// TwinCAT 3 PLC project Plc_CHALET_Xts
// Title: CHALET_Xts
// Company: Beckhoff CH
// ProjectVersion: 4.2.1
// ProgramVersion: 3.1.4023.0
// libraries:
//   CHALET_BaseComponents, * (Beckhoff CH)
//   CHALET_Nc, * (Beckhoff CH)
//   Tc2_EtherCAT, * (Beckhoff Automation GmbH)
//   Tc2_Math, * (Beckhoff Automation GmbH)
//   Tc2_MC2, * (Beckhoff Automation GmbH)
//   Tc2_Standard, * (Beckhoff Automation GmbH)
//   Tc2_System, * (Beckhoff Automation GmbH)
//   Tc3_EventLogger, * (Beckhoff Automation GmbH)
//   Tc3_Mc3Definitions, * (Beckhoff Automation GmbH)
//   Tc3_McCollisionAvoidance, * (Beckhoff Automation GmbH)
//   Tc3_McCoordinatedMotion, * (Beckhoff Automation GmbH)
//   Tc3_Module, * (Beckhoff Automation GmbH)
//   Tc3_XTS_Utility, * (Beckhoff Automation GmbH)
// project tree:
//   COMPENENTs/Casting/ ToMover.TcPOU, ToGroup.TcPOU, ToMover_PLC.TcPOU, ToStation_PLC.TcPOU, ToTrigger.TcPOU, ToEnvironment.TcPOU, ToStation.TcPOU
//   COMPENENTs/ Class Diagram.TcCD (not stored)
//   COMPENENTs/Environment/ FB_XTS_Environment.TcPOU, I_XTS_Environment.TcIO
//   COMPENENTs/Group/ E_NcGroupCommands.TcDUT, FB_XTS_Group.TcPOU, I_XTS_Group.TcIO
//   COMPENENTs/Lubrication/ E_LubricationMode.TcDUT, E_SystemType.TcTLEO, FB_LubricationXTS.TcPOU
//   COMPENENTs/Mover/ FB_XTS_Axis.TcPOU, FB_XTS_Mover.TcPOU, I_XTS_Axis.TcIO, I_XTS_Mover.TcIO, I_XTS_Mover_PLC.TcIO
//   COMPENENTs/Mover/ProductData/ FB_XTS_ProductData.TcPOU, I_XTS_ProductData.TcIO
//   COMPENENTs/Station/ FB_XTS_Station.TcPOU, I_XTS_Station.TcIO, I_XTS_Station_PLC.TcIO
//   COMPENENTs/System/ FB_XTS_System.TcPOU, I_XTS_System_PLC.TcIO, I_XTS_System_Registration.TcIO
//   COMPENENTs/Trigger/ FB_XTS_Trigger.TcPOU, I_XTS_Trigger.TcIO
//   COMPENENTs/Zone/ FB_XTS_Zone.TcPOU, I_XTS_Zone.TcIO
//   Diag/ FB_XtsEtherCatDiag.TcPOU, ST_XtsMotorEtherCatDiag.TcDUT
//   FUNCTIONs/ F_BuildLogString.TcPOU, F_GetDistToPosModulo.TcPOU, F_InLimitTest.TcPOU
//   / XtsParameterlist.TcGVL

// ---- COMPENENTs/Group/E_NcGroupCommands.TcDUT
{attribute 'qualified_only'}
{attribute 'strict'}
{attribute 'to_string'}
TYPE E_NcGroupCommands :
(
	None:=0,
	GroupDisable:=150,
	GroupEnable,
	GroupReset,
	AddAxisListToGroup,
	RemoveAxisFromGroup,
	UngroupAllAxes
);
END_TYPE

// ---- COMPENENTs/Lubrication/E_LubricationMode.TcDUT
{attribute 'qualified_only'}
TYPE E_LubricationMode :
(
	TimeBased,
	DistanceBased,
	Continous
);
END_TYPE

// ---- COMPENENTs/Lubrication/E_SystemType.TcTLEO
{attribute 'qualified_only'}
TYPE E_SystemType :
(
 	BekaPico,
	SkfETP2WZ
);
END_TYPE

// ---- Diag/ST_XtsMotorEtherCatDiag.TcDUT
TYPE ST_XtsMotorEtherCatDiag :
STRUCT
	fbSource : FB_TcSourceInfo;
	fbAlarmNotInOpMode : FB_TcAlarm;
	fbAlarmNoCommunication : FB_TcAlarm;
	
	fbGetSlaveState : FB_EcGetSlaveState;
	nLastState : BYTE;
END_STRUCT
END_TYPE

// ---- XtsParameterlist.TcGVL
{attribute 'qualified_only'}
VAR_GLOBAL CONSTANT
	
	(*Checks whether the TC3 event logger is set as standard in the XTS prosessing unit.*)
	B_MSG_IF_TC3EVENTLOGGER_IS_NOT_DEFAULT: BOOL := TRUE;	

	MAX_MOVER_PER_SYSTEM : UINT := 50;
	MAX_MOTORS_PER_SYSTEM : UINT := 100;
	STATISTIC_AVG_PERIOD : TIME := T#10S;
END_VAR

// ---- COMPENENTs/Environment/I_XTS_Environment.TcIO
INTERFACE I_XTS_Environment  EXTENDS I_CH_Object

{attribute 'monitoring':='call'}
PROPERTY HR : HRESULT
GET
END_GET
END_PROPERTY

METHOD Initialize : HRESULT
END_METHOD

{attribute 'monitoring':='call'}
PROPERTY TrackIsRing : BOOL
GET
END_GET
END_PROPERTY

{attribute 'monitoring':='call'}
PROPERTY TrackLength : LREAL
GET
END_GET
END_PROPERTY

METHOD Update : HRESULT
VAR_INPUT
END_VAR
END_METHOD

PROPERTY UtilityEnvirement : Tc3_XTS_Utility.i_TcIoXtsEnvironment
GET
END_GET
END_PROPERTY

END_INTERFACE

// ---- COMPENENTs/Group/I_XTS_Group.TcIO
INTERFACE I_XTS_Group  EXTENDS I_CH_Object

METHOD AddAxisListToGroup : HRESULT
VAR_INPUT
	ipMovers : I_CH_List;
END_VAR
END_METHOD

METHOD AddingAxisToGroup : HRESULT
END_METHOD

PROPERTY AllAxesStanding : Bool
GET
END_GET
END_PROPERTY

METHOD ChangeGapMode : HRESULT
VAR_INPUT
	bFast : BOOL;
END_VAR
END_METHOD

METHOD Disable : HRESULT
VAR_INPUT
END_VAR
END_METHOD

METHOD Enable : HRESULT
VAR_INPUT
END_VAR
END_METHOD

{attribute 'monitoring':='call'}
PROPERTY GroupEnabled : BOOL
GET
END_GET
END_PROPERTY

{attribute 'monitoring':='call'}
PROPERTY HR : HRESULT
GET
END_GET
END_PROPERTY

METHOD Initialize : HRESULT
VAR_INPUT
END_VAR
END_METHOD

METHOD RemoveAxisFromGroup : HRESULT
VAR_INPUT
	ipMover : I_XTS_Mover;
END_VAR
END_METHOD

METHOD Reset : HRESULT
VAR_INPUT
END_VAR
END_METHOD

METHOD UngroupAllAxes : HRESULT
VAR_INPUT
END_VAR
END_METHOD

METHOD Update : HRESULT
VAR_INPUT
END_VAR
END_METHOD

{attribute 'monitoring':='call'}
PROPERTY UtilityCAGroup : I_Mc2CaGroup
GET
END_GET
END_PROPERTY

END_INTERFACE

// ---- COMPENENTs/Mover/I_XTS_Axis.TcIO
INTERFACE I_XTS_Axis EXTENDS CHALET_Nc.I_NcAxis_PLC

METHOD HaltCA : I_CH_Feedback
VAR_INPUT
	fDeceleration          : LREAL;
    fJerk                  : LREAL;
    fGap                   : LREAL;
END_VAR
END_METHOD

{attribute 'TcRpcEnable':='1'} //call methode via OPC-UA conection
METHOD MoveAbsoluteCA  : I_CH_Feedback
VAR_INPUT
	fPosition		: LREAL;
	
	(* This value determines the minimum gap to the predecessor for Collision Avoidance. *)
	fGap			: LREAL;
	
	(* Use the default dynamics if input=0. 
	The default dynamics can be read and written via property and is initialized with the default values in the NC parameter list. *)
	fVelocity		: LREAL;
	
	(* Use the default dynamics if input=0. 
	The default dynamics can be read and written via property and is initialized with the default values in the NC parameter list. *)
	fAcceleration	: LREAL;
	
	(* Use the default dynamics if input=0. 
	The default dynamics can be read and written via property and is initialized with the default values in the NC parameter list. *)
	fDeceleration	: LREAL;
	
	(* Use the default dynamics if input=0. 
	The default dynamics can be read and written via property and is initialized with the default values in the NC parameter list. *)
	fJerk			: LREAL;
	
	(* Defines the direction of the movement (e.g. for a modulo axis). 
		input=0 = mcDirectionNonModulo*)
	eDirection	: Tc3_Mc3Definitions.MC_DIRECTION;
	
	(* Use the Aborting mode without buffering if input=0. 
	BufferModes:
		-MC_Aborting: Default mode without buffering. The command is executed immediately and interrupts any other command that may be running.
		-MC_Buffered: The command is executed once no other command is running on the axis. The previous movement continues until it has stopped. The following command is started from standstill. *)
	eBufferMode   : Tc3_Mc3Definitions.MC_BUFFER_MODE;
END_VAR
END_METHOD

END_INTERFACE

// ---- COMPENENTs/Mover/I_XTS_Mover.TcIO
INTERFACE I_XTS_Mover EXTENDS I_CH_Object

{attribute 'OPC.UA.DA.Property' := '1'}
{attribute 'monitoring':='call'}
PROPERTY Coupled : BOOL
GET
END_GET
END_PROPERTY

METHOD Disable : HRESULT
VAR_INPUT
END_VAR
END_METHOD

{attribute 'monitoring':='call'}
PROPERTY DrivenDistance : LREAL
GET
END_GET
END_PROPERTY

METHOD Enable : HRESULT
VAR_INPUT
END_VAR
END_METHOD

{attribute 'OPC.UA.DA.Property' := '1'}
{attribute 'monitoring':='call'}
PROPERTY Feedback : I_CH_Feedback
GET
END_GET
END_PROPERTY

PROPERTY getAxisRef : REFERENCE TO Tc2_MC2.AXIS_REF
GET
END_GET
END_PROPERTY

METHOD HaltCA : HRESULT
VAR_INPUT
END_VAR
END_METHOD

{attribute 'monitoring':='call'}
PROPERTY IdentInGroup : IDENT_IN_GROUP_REF
GET
END_GET
END_PROPERTY

{attribute 'monitoring':='call'}
PROPERTY LagDistance : LREAL
GET
END_GET
END_PROPERTY

{attribute 'monitoring':='call'}
PROPERTY LastCmdTargedGap : LREAL
GET
END_GET
END_PROPERTY

{attribute 'monitoring':='call'}
PROPERTY LastCmdTargedPosition : LREAL
GET
END_GET
END_PROPERTY

{attribute 'monitoring':='call'}
PROPERTY LastCmdTargedVelocity : LREAL
GET
END_GET
END_PROPERTY

METHOD MoveAbsCA : HRESULT
VAR_INPUT
    fPosition              : LREAL;
    fVelocity              : LREAL;
    fGap                   : LREAL;
    eDirection             : Tc3_Mc3Definitions.MC_DIRECTION;
END_VAR
END_METHOD

{attribute 'monitoring':='call'}
PROPERTY MoverInGroup : BOOL
GET
END_GET
SET
END_SET
END_PROPERTY

{attribute 'OPC.UA.DA.Property' := '1'}
{attribute 'monitoring':='call'}
PROPERTY Moving : BOOL
GET
END_GET
END_PROPERTY

{attribute 'monitoring':='call'}
PROPERTY NextMover : I_XTS_Mover
GET
END_GET
END_PROPERTY

{attribute 'monitoring':='call'}
PROPERTY OID : OTCID
GET
END_GET
END_PROPERTY

{attribute 'monitoring':='call'}
PROPERTY ParentStation : I_XTS_Station
GET
END_GET
SET
END_SET
END_PROPERTY

{attribute 'monitoring':='call'}
PROPERTY PositionOnTrack : LREAL
GET
END_GET
END_PROPERTY

METHOD Reset : HRESULT
VAR_INPUT
END_VAR
END_METHOD

{attribute 'monitoring':='call'}
PROPERTY SetAcceleration : LREAL
GET
END_GET
END_PROPERTY

{attribute 'monitoring':='call'}
PROPERTY SetVelocity : LREAL
GET
END_GET
END_PROPERTY

{attribute 'monitoring':='call'}
PROPERTY TargedStation : STRING
GET
END_GET
SET
END_SET
END_PROPERTY

{attribute 'monitoring':='call'}
PROPERTY UtilityMover : I_TcIoXtsXpuMover
GET
END_GET
END_PROPERTY

END_INTERFACE

// ---- COMPENENTs/Mover/I_XTS_Mover_PLC.TcIO
INTERFACE I_XTS_Mover_PLC EXTENDS I_CH_Object

{attribute 'OPC.UA.DA.Property' := '1'}
{attribute 'monitoring':='call'}
PROPERTY DefaultAcceleration : LREAL
GET
END_GET
SET
END_SET
END_PROPERTY

{attribute 'OPC.UA.DA.Property' := '1'}
{attribute 'monitoring':='call'}
PROPERTY DefaultDeceleration : LREAL
GET
END_GET
SET
END_SET
END_PROPERTY

{attribute 'OPC.UA.DA.Property' := '1'}
{attribute 'monitoring':='call'}
PROPERTY DefaultJerk : LREAL
GET
END_GET
SET
END_SET
END_PROPERTY

{attribute 'monitoring':='call'}
PROPERTY DrivenDistance : LREAL
GET
END_GET
END_PROPERTY

(*The _ PLC interface provides the user with a simplified interface for commanding between the stations. Sometimes, however, this is not enough. 
Either you get the corresponding interface with the __Queryinterface or you can get full access with this property.*)
PROPERTY FullAccess : I_XTS_Mover
GET
END_GET
END_PROPERTY

{attribute 'monitoring':='call'}
PROPERTY LagDistance : LREAL
GET
END_GET
END_PROPERTY

{attribute 'monitoring':='call'}
PROPERTY LastCmdTargedGap : LREAL
GET
END_GET
END_PROPERTY

{attribute 'monitoring':='call'}
PROPERTY LUID : STRING
GET
END_GET
END_PROPERTY

//Returns the ID of the mover.
{attribute 'monitoring':='call'}
PROPERTY MoverID : STRING(3)
GET
END_GET
END_PROPERTY

{attribute 'monitoring':='call'}
PROPERTY NameXtsMover : STRING
GET
END_GET
END_PROPERTY

{attribute 'monitoring':='call'}
//Interface to the underlying NC axis object. Not all commands may be compatible with the CA group
PROPERTY NcAxis : I_XTS_Axis
GET
END_GET
END_PROPERTY

{attribute 'monitoring':='call'}
PROPERTY PositionOnTrack : LREAL
GET
END_GET
END_PROPERTY

{attribute 'monitoring':='call'}
PROPERTY PUBLIC ProductData : I_XTS_ProductData
GET
END_GET
SET
END_SET
END_PROPERTY

{attribute 'monitoring':='call'}
PROPERTY SetVelocity : LREAL
GET
END_GET
END_PROPERTY

{attribute 'monitoring':='call'}
PROPERTY TargedStation : STRING
GET
END_GET
END_PROPERTY

{attribute 'monitoring':='call'}
PROPERTY UtilityMover : I_TcIoXtsXpuMover
GET
END_GET
END_PROPERTY

END_INTERFACE

// ---- COMPENENTs/Mover/ProductData/I_XTS_ProductData.TcIO
INTERFACE I_XTS_ProductData EXTENDS __SYSTEM.IQueryInterface

{attribute 'monitoring':='call'}
PROPERTY LinkedMover : I_XTS_Mover_PLC
GET
END_GET
END_PROPERTY

METHOD LinkToMover : BOOL //it is not necessary to call this method. This is already done internally
VAR_INPUT
	ipMoverPlc : I_XTS_Mover_PLC;
END_VAR
END_METHOD

END_INTERFACE

// ---- COMPENENTs/Station/I_XTS_Station.TcIO
INTERFACE I_XTS_Station EXTENDS I_CH_Object

METHOD AddMoverToQueue : HRESULT
VAR_INPUT
	ipMover : I_XTS_Mover;
END_VAR
END_METHOD

//Call this Methode whith seq 0->99, and wait each step until S_OK is returned
METHOD Configure : HRESULT
VAR_INPUT
	nSeq : UINT; //0->100
END_VAR
END_METHOD

{attribute 'monitoring':='call'}
PROPERTY CtsEmptySpaceInQueue : UDINT
GET
END_GET
END_PROPERTY

{attribute 'monitoring':='call'}
PROPERTY CtsMoversInQueue : UDINT
GET
END_GET
END_PROPERTY

METHOD DeleteMoversQueue : HRESULT
VAR_INPUT
END_VAR
END_METHOD

{attribute 'monitoring':='call'}
PROPERTY HR : HRESULT
GET
END_GET
END_PROPERTY

{attribute 'monitoring':='call'}
PROPERTY LUID : STRING
GET
END_GET
END_PROPERTY

{attribute 'monitoring':='call'}
PROPERTY MoverGapAtExit : LREAL
GET
END_GET
SET
END_SET
END_PROPERTY

{attribute 'monitoring':='call'}
PROPERTY MoverQueueSize : UINT
GET
END_GET
SET
END_SET
END_PROPERTY

{attribute 'monitoring':='call'}
PROPERTY MoversInPlace : BOOL
GET
END_GET
END_PROPERTY

{attribute 'monitoring':='call'}
PROPERTY MoversInQueue : REFERENCE TO ARRAY [0..(XtsParameterlist.MAX_MOVER_PER_SYSTEM-1)] OF I_XTS_Mover_PLC // Return a sorted list of movers in this zone. Index 0 is the mover in Front.
GET
END_GET
END_PROPERTY

{attribute 'monitoring':='call'}
PROPERTY MoverVelocityAtExit : LREAL
GET
END_GET
SET
END_SET
END_PROPERTY

{attribute 'monitoring':='call'}
PROPERTY PositionOnTrack : LREAL
GET
END_GET
END_PROPERTY

{attribute 'monitoring':='call'}
PROPERTY ReadyToRecvMovers : BOOL
GET
END_GET
SET
END_SET
END_PROPERTY

METHOD SendMoversToStation : HRESULT
VAR_INPUT
	sTargedStation : STRING;
END_VAR
END_METHOD

{attribute 'monitoring':='call'}
PROPERTY StationsAhead : I_XTS_Station
GET
END_GET
END_PROPERTY

END_INTERFACE

// ---- COMPENENTs/Station/I_XTS_Station_PLC.TcIO
INTERFACE I_XTS_Station_PLC EXTENDS I_CH_Object

METHOD ChangePos : HRESULT
VAR_INPUT
	fNewPosOnTrack : LREAL;
END_VAR
END_METHOD

(*The _ PLC interface provides the user with a simplified interface for commanding between the stations. Sometimes, however, this is not enough. 
Either you get the corresponding interface with the __Queryinterface or you can get full access with this property.*)
PROPERTY FullAccess : I_XTS_Station
GET
END_GET
END_PROPERTY

{attribute 'monitoring':='call'}
PROPERTY LUID : STRING
GET
END_GET
END_PROPERTY

{attribute 'monitoring':='call'}
PROPERTY MoverQueueSize : UINT
GET
END_GET
SET
END_SET
END_PROPERTY

{attribute 'monitoring':='call'}
PROPERTY MoversInPlace : BOOL
GET
END_GET
END_PROPERTY

{attribute 'monitoring':='call'}
PROPERTY MoversInQueue : REFERENCE TO ARRAY [0..(XtsParameterlist.MAX_MOVER_PER_SYSTEM-1)] OF I_XTS_Mover_PLC // Return a sorted list of movers in this zone. Index 0 is the mover in Front.
GET
END_GET
END_PROPERTY

{attribute 'monitoring':='call'}
PROPERTY MoverVelocityAtExit : LREAL //[mm/s] Every mover that leaves or passes the station gets this new velocity as a target.
GET
END_GET
SET
END_SET
END_PROPERTY

{attribute 'monitoring':='call'}
PROPERTY PositionOnTrack : LREAL
GET
END_GET
END_PROPERTY

{attribute 'monitoring':='call'}
PROPERTY ProcessSimulationActive : BOOL
GET
END_GET
END_PROPERTY

{attribute 'monitoring':='call'}
//prevent further movers from entering the station, 
//e.g. to prevent a collision. All movers that are already moving to reach this station will be stopped with a stop 
//and restarted with Ready True.
PROPERTY ReadyToRecvMovers : BOOL
GET
END_GET
SET
END_SET
END_PROPERTY

METHOD SendMoversToStation : HRESULT
VAR_INPUT
	sTargedStation : STRING;
END_VAR
END_METHOD

//If a valid time (>0seconds) is set and the configured destination station exists, then the movers will be sent away automatically after this time from now on.
METHOD SimulationStart : HRESULT
VAR_INPUT
	fProcessDuration 	: LREAL; //[s]
	sTargedStation		: STRING; //LUID of the targed station to automatic send after the duration
END_VAR
END_METHOD

//If a valid time (>0seconds) is set and the configured destination station exists, then the movers will be sent away automatically after this time from now on.
METHOD SimulationStartEx : HRESULT
VAR_INPUT
	fProcessDuration 		: LREAL; //[s]
	ipStation				: I_Xts_Station_PLC; //unique station to automatic send after the duration
END_VAR
END_METHOD

METHOD SimulationStop : HRESULT
END_METHOD

{attribute 'monitoring':='call'}
PROPERTY SuppressDynamicsChange : BOOL
GET
END_GET
SET
END_SET
END_PROPERTY

{attribute 'monitoring':='call'}
//A time that is waited as soon as the mover is in the station (including the monitoring window) before “MoversInPlace” is set. e.g. used to stabilize the workpiece
PROPERTY TargetPosMonitoringTime : TIME
GET
END_GET
SET
END_SET
END_PROPERTY

{attribute 'monitoring':='call'}
//How many mm before the mover reaches the position is “MoversInPlace” set for the process. 
//This distance can also be set very large (e.g. 100mm) for moving past without stopping.
PROPERTY TargetPosWindow : LREAL
GET
END_GET
SET
END_SET
END_PROPERTY

END_INTERFACE

// ---- COMPENENTs/System/I_XTS_System_PLC.TcIO
INTERFACE I_XTS_System_PLC EXTENDS I_CH_Object

METHOD Disable : I_CH_Feedback
VAR_INPUT
END_VAR
END_METHOD

{attribute 'monitoring':='call'}
PROPERTY Disabled : Bool
GET
END_GET
END_PROPERTY

METHOD Enable : I_CH_Feedback
VAR_INPUT
END_VAR
END_METHOD

{attribute 'monitoring':='call'}
PROPERTY Enabled : Bool
GET
END_GET
END_PROPERTY

{attribute 'monitoring':='call'}
PROPERTY Feedback : CHALET_BaseComponents.I_CH_Feedback
GET
END_GET
END_PROPERTY

METHOD Initialize : HRESULT
VAR_INPUT
END_VAR
END_METHOD

{attribute 'monitoring':='call'}
PROPERTY Initialized : BOOL
GET
END_GET
END_PROPERTY

METHOD Reset : HRESULT
VAR_INPUT
END_VAR
END_METHOD

METHOD Station : I_XTS_Station_PLC
VAR_INPUT
	sLUID : STRING;
END_VAR
END_METHOD

PROPERTY SuppressAllDynamicsChanges : BOOL
SET
END_SET
END_PROPERTY

{attribute 'monitoring':='call'}
PROPERTY TrackLength : LREAL
GET
END_GET
END_PROPERTY

METHOD Update : HRESULT
VAR_INPUT
END_VAR
END_METHOD

END_INTERFACE

// ---- COMPENENTs/System/I_XTS_System_Registration.TcIO
INTERFACE I_XTS_System_Registration

{attribute 'monitoring':='call'}
PROPERTY Disabled : Bool
GET
END_GET
END_PROPERTY

{attribute 'monitoring':='call'}
PROPERTY Enabled : Bool
GET
END_GET
END_PROPERTY

{attribute 'monitoring':='call'}
PROPERTY Environment : I_XTS_Environment
GET
END_GET
END_PROPERTY

METHOD getMoverInFront : I_Xts_Mover
VAR_INPUT
	ipMover : I_Xts_Mover;
END_VAR
END_METHOD

{attribute 'monitoring':='call'}
PROPERTY Initialized : BOOL
GET
END_GET
END_PROPERTY

METHOD LinkEnvironment : HRESULT
VAR_INPUT
	ipEnvironment : CHALET_BaseComponents.I_CH_Object;
END_VAR
END_METHOD

METHOD LinkGroup : HRESULT
VAR_INPUT
	ipGroup : CHALET_BaseComponents.I_CH_Object;
END_VAR
END_METHOD

{attribute 'monitoring':='call'}
PROPERTY Movers : CHALET_BaseComponents.I_CH_LIST
GET
END_GET
END_PROPERTY

METHOD RegisterMover : HRESULT
VAR_INPUT
	ipMover : CHALET_BaseComponents.I_CH_Object;
END_VAR
END_METHOD

METHOD RegisterStation : HRESULT
VAR_INPUT
	ipStation : CHALET_BaseComponents.I_CH_Object;
END_VAR
END_METHOD

METHOD RegisterTrigger : HRESULT
VAR_INPUT
	ipTrigger	: CHALET_BaseComponents.I_CH_Object;
END_VAR
END_METHOD

METHOD RegisterZone : HRESULT
VAR_INPUT
	ipZone	: CHALET_BaseComponents.I_CH_Object;
END_VAR
END_METHOD

PROPERTY Stations : I_CH_LIST
GET
END_GET
END_PROPERTY

{attribute 'monitoring':='call'}
PROPERTY TrackLength : LREAL
GET
END_GET
END_PROPERTY

END_INTERFACE

// ---- COMPENENTs/Trigger/I_XTS_Trigger.TcIO
INTERFACE I_XTS_Trigger  EXTENDS I_CH_Object

{attribute 'monitoring':='call'}
PROPERTY HR : HRESULT
GET
END_GET
END_PROPERTY

PROPERTY ListOfMoversToCheck : I_CH_List
SET
END_SET
END_PROPERTY

{attribute 'monitoring':='call'}
PROPERTY MoverAtTrigger : I_XTS_Mover
GET
END_GET
END_PROPERTY

{attribute 'monitoring':='call'}
PROPERTY MoverDetected : BOOL
GET
END_GET
END_PROPERTY

{attribute 'monitoring':='call'}
PROPERTY PositionOnTrack : LREAL
GET
END_GET
SET
END_SET
END_PROPERTY

{attribute 'monitoring':='call'}
PROPERTY TimeStamp : T_DCTIME64;
GET
END_GET
END_PROPERTY

{attribute 'monitoring':='call'}
PROPERTY TriggerDirection : Tc2_MC2.MC_Direction
GET
END_GET
SET
END_SET
END_PROPERTY

END_INTERFACE

// ---- COMPENENTs/Zone/I_XTS_Zone.TcIO
INTERFACE I_XTS_Zone  EXTENDS I_CH_Object

{attribute 'monitoring':='call'}
PROPERTY CtsMoversInZone : UINT
GET
END_GET
END_PROPERTY

{attribute 'monitoring':='call'}
PROPERTY EndPositionOnTrack : LREAL
GET
END_GET
SET
END_SET
END_PROPERTY

{attribute 'monitoring':='call'}
PROPERTY HR : HRESULT
GET
END_GET
END_PROPERTY

PROPERTY ListOfMoversToCheck : I_CH_List
SET
END_SET
END_PROPERTY

{attribute 'monitoring':='call'}
PROPERTY MoversInZone : REFERENCE TO ARRAY [0..(XtsParameterlist.MAX_MOVER_PER_SYSTEM-1)] OF I_XTS_Mover_PLC
GET
END_GET
END_PROPERTY

{attribute 'monitoring':='call'}
PROPERTY StartPositionOnTrack : LREAL
GET
END_GET
SET
END_SET
END_PROPERTY

END_INTERFACE

// ---- COMPENENTs/Casting/ToMover.TcPOU
FUNCTION ToMover : BOOL
VAR_INPUT
	ipChObject : I_CH_OBJECT;
	ipXtsMover : REFERENCE TO I_XTS_Mover;
END_VAR

VAR
	ipTmp : I_XTS_Mover;
END_VAR

(* 
   1. Test if the interface exists
   2. Test if the object implements a "Object" interface 
   3. Write reference to interface in parameter
   4. Returne TRUE if succesfull
*)
IF ipChObject <> 0 AND_THEN __QUERYINTERFACE(ipChObject,ipTmp) THEN
	ipXtsMover := ipTmp;
	ToMover := TRUE;
END_IF

END_FUNCTION

// ---- COMPENENTs/Casting/ToGroup.TcPOU
FUNCTION ToGroup : BOOL
VAR_INPUT
	ipChObject : I_CH_OBJECT;
	ipXtsGroup : REFERENCE TO I_XTS_Group;
END_VAR

VAR
	ipTmp : I_XTS_Group;
END_VAR

(* 
   1. Test if the interface exists
   2. Test if the object implements a "Object" interface 
   3. Write reference to interface in parameter
   4. Returne TRUE if succesfull
*)
IF ipChObject <> 0 AND_THEN __QUERYINTERFACE(ipChObject,ipTmp) THEN
	ipXtsGroup := ipTmp;
	ToGroup := TRUE;
END_IF

END_FUNCTION

// ---- COMPENENTs/Casting/ToMover_PLC.TcPOU
FUNCTION ToMover_PLC : BOOL
VAR_INPUT
	ipChObject : I_CH_OBJECT;
	ipXtsMover : REFERENCE TO I_XTS_Mover_PLC;
END_VAR

VAR
	ipTmp : I_XTS_Mover_PLC;
END_VAR

(* 
   1. Test if the interface exists
   2. Test if the object implements a "Object" interface 
   3. Write reference to interface in parameter
   4. Returne TRUE if succesfull
*)
IF ipChObject <> 0 AND_THEN __QUERYINTERFACE(ipChObject,ipTmp) THEN
	ipXtsMover := ipTmp;
	ToMover_PLC := TRUE;
END_IF

END_FUNCTION

// ---- COMPENENTs/Casting/ToStation_PLC.TcPOU
FUNCTION ToStation_PLC : BOOL
VAR_INPUT
	ipChObject : I_CH_OBJECT;
	ipXtsStationPLC : REFERENCE TO I_XTS_Station_PLC;
END_VAR

VAR
	ipTmp : I_XTS_Station_PLC;
END_VAR

(* Register the Station
   1. Test if the interface exists
   2. Test if the object implements a "Object" interface 
*)
IF ipChObject <> 0 AND_THEN __QUERYINTERFACE(ipChObject,ipTmp) THEN
	ipXtsStationPLC := ipTmp;
	ToStation_PLC := TRUE;
END_IF

END_FUNCTION

// ---- COMPENENTs/Casting/ToTrigger.TcPOU
FUNCTION ToTrigger : BOOL
VAR_INPUT
	ipChObject : I_CH_OBJECT;
	ipXtsTrigger : REFERENCE TO I_XTS_Trigger;
END_VAR

VAR
	ipTmp : I_XTS_Trigger;
END_VAR

(* 
   1. Test if the interface exists
   2. Test if the object implements a "Object" interface 
   3. Write reference to interface in parameter
   4. Returne TRUE if succesfull
*)
IF ipChObject <> 0 AND_THEN __QUERYINTERFACE(ipChObject,ipTmp) THEN
	ipXtsTrigger := ipTmp;
	ToTrigger := TRUE;
END_IF

END_FUNCTION

// ---- COMPENENTs/Casting/ToEnvironment.TcPOU
FUNCTION ToEnvironment : BOOL
VAR_INPUT
	ipChObject : I_CH_OBJECT;
	ipXtsEnvironment : REFERENCE TO I_XTS_Environment;
END_VAR

VAR
	ipTmp : I_XTS_Environment;
END_VAR

(* 
   1. Test if the interface exists
   2. Test if the object implements a "Object" interface 
   3. Write reference to interface in parameter
   4. Returne TRUE if succesfull
*)
IF ipChObject <> 0 AND_THEN __QUERYINTERFACE(ipChObject,ipTmp) THEN
	ipXtsEnvironment := ipTmp;
	ToEnvironment := TRUE;
END_IF

END_FUNCTION

// ---- COMPENENTs/Casting/ToStation.TcPOU
FUNCTION ToStation : BOOL
VAR_INPUT
	ipChObject : I_CH_OBJECT;
	ipXtsStation : REFERENCE TO I_XTS_Station;
END_VAR

VAR
	ipTmp : I_XTS_Station;
END_VAR

(* Register the Station
   1. Test if the interface exists
   2. Test if the object implements a "Object" interface 
*)
IF ipChObject <> 0 AND_THEN __QUERYINTERFACE(ipChObject,ipTmp) THEN
	ipXtsStation := ipTmp;
	ToStation := TRUE;
END_IF

END_FUNCTION

// ---- COMPENENTs/Environment/FB_XTS_Environment.TcPOU
{attribute 'no_explicit_call' := 'Do not call the body - Stick to OOP'}
FUNCTION_BLOCK FB_XTS_Environment EXTENDS FB_CH_Object IMPLEMENTS I_XTS_Environment
VAR
	{attribute 'hide'}
	bInitDone : BOOL ;
	{attribute 'hide'}
	ipXtsSystem : I_XTS_System_Registration;

	fbUtilityEnvironment : Tc3_XTS_Utility.FB_TcIoXtsEnvironment;
	
	//Ethercat Diagnostic of all XTS Motors
	fbXtsEtherCatDiag		: FB_XtsEtherCatDiag(	ipUtilityEnvironmentv 				:=  fbUtilityEnvironment,
													bCheckIfTc3EventloggerIsSelected 	:= XtsParameterlist.B_MSG_IF_TC3EVENTLOGGER_IS_NOT_DEFAULT);
	
	{attribute 'hide'}
	fbXtsEnvironmentVisu : Tc3_XTS_Utility.FB_XtsEnvironmentVisu;
		
END_VAR

METHOD FB_init : BOOL
VAR_INPUT
	bInitRetains : BOOL; // if TRUE, the retain variables are initialized (warm start / cold start)
	bInCopyCode : BOOL;  // if TRUE, the instance afterwards gets moved into the copy code (online change)

	ipXtsSystem : I_XTS_System_Registration; //Interface to XTS system object	
END_VAR
VAR_INST
	{attribute 'hide'}
	bFBInitCalledOnce : BOOL; //Do the following code once during start up and not during onlinechange
END_VAR
//Do the following code once during start up and not during onlinechange
IF NOT bFBInitCalledOnce THEN 
	
	//Regristrate object in System
	IF ipXtsSystem <> 0 THEN
		ipXtsSystem.LinkEnvironment(THIS^);
		THIS^.ipXtsSystem := ipXtsSystem;
	END_IF



END_IF

bFBInitCalledOnce := TRUE;
END_METHOD

{warning 'add property implementation'}
{attribute 'monitoring':='call'}
PROPERTY HR : HRESULT
GET
HR := S_OK;
END_GET
END_PROPERTY

METHOD Initialize : HRESULT
VAR 
	hr : HRESULT;
END_VAR
IF NOT THIS^.bInitDone THEN
	Initialize := S_PENDING;	

	//Enable init Info Server if needed
	fbUtilityEnvironment.P_XtsEnvironmentConfiguration.bEnableInitInfoServer := TRUE;

	//Enable init CA Group if needed
	fbUtilityEnvironment.P_XtsEnvironmentConfiguration.bEnableInitCaGroup := TRUE;

	IF NOT fbUtilityEnvironment.P_IsInitialized THEN	
		//Start init
		fbUtilityEnvironment.Init(bExecute := TRUE); 
		hr := GetMostSignificant(hr, S_PENDING);	
 	ELSE
		//Stop init
		fbUtilityEnvironment.Init(bExecute := FALSE);
	END_IF
	
	// Link data Pointer 
	fbXtsEnvironmentVisu(ipTcIoXtsEnvironment:=UtilityEnvirement);

	// Ethercat Diagnostic of all XTS Motors
	hr := GetMostSignificant(hr, fbXtsEtherCatDiag.Initialize());
	

	THIS^.bInitDone  :=  hr = S_OK;
END_IF

Initialize := hr;
END_METHOD

{attribute 'monitoring':='call'}
PROPERTY TrackIsRing : BOOL
GET
IF fbUtilityEnvironment.P_IsInitialized THEN
	TrackIsRing := fbUtilityEnvironment.Mc2CaGroup(1).GetRailIsRing();
END_IF
END_GET
END_PROPERTY

{attribute 'monitoring':='call'}
PROPERTY TrackLength : LREAL
GET
IF fbUtilityEnvironment.P_IsInitialized THEN
	TrackLength := fbUtilityEnvironment.Mc2CaGroup(1).GetRailLength();
END_IF
END_GET
END_PROPERTY

METHOD Update : HRESULT
VAR
	hr : HRESULT;
END_VAR

fbXtsEtherCatDiag.Update();

fbXtsEnvironmentVisu.Cycle();

Update:= hr;
END_METHOD

PROPERTY UtilityEnvirement : Tc3_XTS_Utility.I_TcIoXtsEnvironment
GET
//Interface to envirement
UtilityEnvirement := fbUtilityEnvironment;
END_GET
END_PROPERTY

END_FUNCTION_BLOCK

// ---- Diag/FB_XtsEtherCatDiag.TcPOU
{attribute 'no_explicit_call' := 'Do not call the body - Stick to OOP'}
(* This FB generates an array with all XTS motor modules. These are now checked cyclically one after the other to see whether the EtherCAT slave controller is in OP mode *)
FUNCTION_BLOCK FB_XtsEtherCatDiag EXTENDS CHALET_BaseComponents.FB_CH_Object
VAR
	ipUtilityEnvironmentv : Tc3_XTS_Utility.I_TcIoXtsEnvironment;
	bCheckIfTc3EventloggerIsSelected : BOOL;
	stMotorDiag : ARRAY[0..N_MAX_CTS_MOTORMODULES-1] OF ST_XtsMotorEtherCatDiag;
	bInitDone : BOOL;
	nIdxTrigger : UINT;
	nCtnMotorModules : UINT;
	fbMsgWrongEventlogger : FB_TcMessage;
	bEventLoggerChecked : BOOL;
END_VAR

VAR CONSTANT
	N_MAX_CTS_MOTORMODULES : UINT := XtsParameterlist.MAX_MOTORS_PER_SYSTEM;
END_VAR

METHOD FB_init : BOOL
VAR_INPUT
	bInitRetains : BOOL; // if TRUE, the retain variables are initialized (warm start / cold start)
	bInCopyCode : BOOL;  // if TRUE, the instance afterwards gets moved into the copy code (online change)
	
	ipUtilityEnvironmentv : Tc3_XTS_Utility.I_TcIoXtsEnvironment;
	
	//Message if TC3_Eventlogger is not set as Eventlogger. Not possible to change online.
	//Must be adjusted in the following object: XtsProcessingUnit/Parameter(Init)/Diagnostic/UsedEventLogger 
	bCheckIfTc3EventloggerIsSelected : BOOL;
END_VAR

VAR
	fbGetCurTaskIdx  : GETCURTASKINDEX;
END_VAR

THIS^.ipUtilityEnvironmentv := ipUtilityEnvironmentv;
THIS^.bCheckIfTc3EventloggerIsSelected := bCheckIfTc3EventloggerIsSelected;
END_METHOD

METHOD Initialize : HRESULT
VAR
	ipObject : ITComObject;
	sObjectName : STRING;
	nIdx, nIdxXpu, nIdxPart, nIdxModule : UINT;
END_VAR
VAR_INST

END_VAR
//Validate interface
IF ipUtilityEnvironmentv = 0 THEN
	Initialize := E_FAIL;
	RETURN;
END_IF

//Wait for an valide XpuCount. At beginn, count is 0
IF ipUtilityEnvironmentv.P_XpuCount = 0 THEN
	Initialize := S_PENDING;;
	RETURN;
END_IF

//Wait for init done
FOR nIdxXpu := 1 TO TO_UINT(ipUtilityEnvironmentv.P_XpuCount)  DO
	IF NOT ipUtilityEnvironmentv.XpuTcIo(nIdxXpu).P_IsInitialized THEN
		Initialize := S_PENDING;;
		RETURN;
	END_IF
END_FOR

//Message if TC3_Eventlogger is not set as Eventlogger. Not possible to change online.
//Must be adjusted in the following object: XtsProcessingUnit/Parameter(Init)/Diagnostic/UsedEventLogger 
IF NOT bEventLoggerChecked  AND THIS^.bCheckIfTc3EventloggerIsSelected THEN
	FOR nIdxXpu := 1 TO TO_UINT(ipUtilityEnvironmentv.P_XpuCount) DO
		IF ipUtilityEnvironmentv.XpuTcIo(nIdxXpu).GetUsedEventLogger() <> EventMessenger.TC3EventLogger THEN
			fbMsgWrongEventlogger.CreateEx(stEventEntry:=TC_EVENTS.CHALET_XTS_Events.TC3EventloggerCheck, ipSourceInfo := THIS^.fbSourceInfo);
			fbMsgWrongEventlogger.Send(0);
			EXIT;
		END_IF
	END_FOR
END_IF
bEventLoggerChecked := TRUE;



//For all Modul in all Parts in all Processing-Units
nIdx := 0;
FOR nIdxXpu := 1 TO TO_UINT(ipUtilityEnvironmentv.P_XpuCount) DO
	FOR nIdxPart := 1 TO ipUtilityEnvironmentv.XpuTcIo(nIdxXpu).P_PartCount DO
		FOR nIdxModule := 1 TO ipUtilityEnvironmentv.XpuTcIo(nIdxXpu).PartTcIo(nIdxPart).P_ModuleCount DO
			//Error, array is to small
			IF (nIdx > (N_MAX_CTS_MOTORMODULES-1)) THEN
				Initialize := E_FAIL;
				RETURN;
			END_IF
			
			//Read object name of motor module
			FW_ObjMgr_GetObjectInstance(oid:= ipUtilityEnvironmentv.XpuTcIo(nIdxXpu).PartTcIo(nIdxPart).ModuleTcIo(nIdxModule).GetMotorTerminalOid() , iid:= TC_GLOBAL_IID_LIST.IID_ITComObject, pipUnk:= ADR(ipObject));
			//Read Name of object if interafce is valid
			IF ipObject <> 0 AND_THEN (ipObject.TcGetObjectName(ADR(sObjectName), SIZEOF(sObjectName)) = S_OK) THEN
				//Set source name + Modulename
				stMotorDiag[nIdx].fbSource.sName := '';
				stMotorDiag[nIdx].fbSource.ExtendName(sObjectName);
				stMotorDiag[nIdx].fbSource.ExtendName(' Part:');
				stMotorDiag[nIdx].fbSource.ExtendName(TO_STRING(nIdxPart));
				stMotorDiag[nIdx].fbSource.ExtendName(' Module:');
				stMotorDiag[nIdx].fbSource.ExtendName(TO_STRING(nIdxModule));	
				ipObject.TcRelease();
			ELSE
				//Set source name
				stMotorDiag[nIdx].fbSource.sName := '';
				stMotorDiag[nIdx].fbSource.ExtendName('Part:');
				stMotorDiag[nIdx].fbSource.ExtendName(TO_STRING(nIdxPart));
				stMotorDiag[nIdx].fbSource.ExtendName(' Module:');
				stMotorDiag[nIdx].fbSource.ExtendName(TO_STRING(nIdxModule));	
			END_IF
			

		
			//Create alarm
			stMotorDiag[nIdx].fbAlarmNotInOpMode.CreateEx(
					stEventEntry := TC_EVENTS.CHALET_XTS_Events.EtherCatSlaveNotInOpMode, 
					ipSourceInfo := stMotorDiag[nIdx].fbSource, 
					bWithConfirmation := FALSE);
					
			stMotorDiag[nIdx].fbAlarmNoCommunication.CreateEx(	
					stEventEntry:= TC_EVENTS.CHALET_XTS_Events.NoCommunication,
					ipSourceInfo 	:= stMotorDiag[nIdx].fbSource, 
					bWithConfirmation := FALSE);
					
			//store ADS conncetion info
			stMotorDiag[nIdx].fbGetSlaveState.sNetId := ipUtilityEnvironmentv.XpuTcIo(nIdxXpu).PartTcIo(nIdxPart).ModuleTcIo(nIdxModule).CoE.AmsNetId;
			stMotorDiag[nIdx].fbGetSlaveState.nSlaveAddr := ipUtilityEnvironmentv.XpuTcIo(nIdxXpu).PartTcIo(nIdxPart).ModuleTcIo(nIdxModule).GetDriveAddress();		

			nIdx := nIdx +1;	
			THIS^.nCtnMotorModules := nIdx;
		END_FOR
	END_FOR
END_FOR
bInitDone := TRUE;
Initialize := S_OK;;
END_METHOD

{attribute 'monitoring':='call'}
PROPERTY Initialized : BOOL
GET
Initialized := bInitDone;
END_GET
END_PROPERTY

METHOD Update : HRESULT
VAR
	nIdx : UINT;
	bErrorNoCom : BOOL;
	bInOpMode : BOOL;
	bReadOfStateFailed : BOOL;
END_VAR
// Force to do init
IF NOT THIS^.bInitDone THEN
	Initialize();
	RETURN;
END_IF


//Trigger each plc cycle 1 read of the motor ethercat slave state - if not allready busy
IF NOT stMotorDiag[nIdxTrigger].fbGetSlaveState.bBusy THEN
	stMotorDiag[nIdxTrigger].fbGetSlaveState(bExecute := TRUE);
	stMotorDiag[nIdxTrigger].fbGetSlaveState(bExecute := FALSE);
	nIdxTrigger := (nIdxTrigger + 1)MOD THIS^.nCtnMotorModules;
END_IF



//For all FBs
FOR nIdx := 0 TO (THIS^.nCtnMotorModules-1) DO
	(*	0x___1 = Slave in 'INIT' state
		0x___2 = Slave in 'PREOP' state
		0x___3 = Slave in 'BOOT' state
		0x___4 = Slave in 'SAFEOP' state
		0x___8 = Slave in 'OP' state		*)
		
		
	//Write Ethercat linkState in TC3 Eventlogger
	bErrorNoCom := (stMotorDiag[nIdx].fbGetSlaveState.state.linkState = 16#01(*NotPresent*));
	IF (NOT bErrorNoCom AND stMotorDiag[nIdx].fbAlarmNoCommunication.bRaised) THEN
		//No error - Reset	
		stMotorDiag[nIdx].fbAlarmNoCommunication.Clear(0,0);
	ELSIF (bErrorNoCom AND NOT stMotorDiag[nIdx].fbAlarmNoCommunication.bRaised) THEN
		//New Error - Raise
		stMotorDiag[nIdx].fbAlarmNoCommunication.ipArguments.Clear();
		stMotorDiag[nIdx].fbAlarmNoCommunication.Raise(0);
	ELSE
		//Alarm is already active
		;
	END_IF	

		
	//Re-Raise alarm on change of state if ethercatslave is not in OP-Mode - Clear if NoCommunication is raised
	bInOpMode := (stMotorDiag[nIdx].fbGetSlaveState.state.deviceState = 16#08(*OP*));
	bReadOfStateFailed := ((stMotorDiag[nIdx].fbGetSlaveState.state.deviceState AND 16#0F(*Mask values 0-15*)) = 16#00);
	IF ((bInOpMode OR bErrorNoCom OR bReadOfStateFailed) AND stMotorDiag[nIdx].fbAlarmNotInOpMode.bRaised) THEN
		//No error - Reset	
		stMotorDiag[nIdx].fbAlarmNotInOpMode.Clear(0,0);
		
	ELSIF (bInOpMode OR bErrorNoCom OR bReadOfStateFailed) THEN
		; //Do nothing
		
	ELSIF (stMotorDiag[nIdx].fbGetSlaveState.state.deviceState <> stMotorDiag[nIdx].nLastState) THEN
		//New Error - Reset, Create and Raise
		stMotorDiag[nIdx].fbAlarmNotInOpMode.Clear(0,0);
		CASE (stMotorDiag[nIdx].fbGetSlaveState.state.deviceState AND 16#0F(*Mask values 0-15*)) OF
			1:  stMotorDiag[nIdx].fbAlarmNotInOpMode.ipArguments.Clear().AddString('INIT'); 	
			2:  stMotorDiag[nIdx].fbAlarmNotInOpMode.ipArguments.Clear().AddString('PREOP');	
			3:  stMotorDiag[nIdx].fbAlarmNotInOpMode.ipArguments.Clear().AddString('BOOT');		
			4:  stMotorDiag[nIdx].fbAlarmNotInOpMode.ipArguments.Clear().AddString('SAFEOP');	
		END_CASE
		stMotorDiag[nIdx].fbAlarmNotInOpMode.Raise(0);
		
	ELSE
		//Alarm is already active
		;
	END_IF
	stMotorDiag[nIdx].nLastState := stMotorDiag[nIdx].fbGetSlaveState.state.deviceState;

	
	//Call cyclic fb
	stMotorDiag[nIdx].fbGetSlaveState();
END_FOR
END_METHOD

END_FUNCTION_BLOCK

// ---- COMPENENTs/Group/FB_XTS_Group.TcPOU
{attribute 'no_explicit_call' := 'Do not call the body - Stick to OOP'}
FUNCTION_BLOCK FB_XTS_Group EXTENDS FB_CH_Object IMPLEMENTS I_XTS_Group
VAR
	{attribute 'hide'}	
	bInitDone : BOOL;
	{attribute 'hide'}
	ipXtsSystem 		: I_XTS_System_Registration;
	{attribute 'hide'}
	ipUtilityCAGroup 	: I_Mc2CaGroup;
	{attribute 'hide'}
	fbAddAxisToGroup 	: Tc3_McCoordinatedMotion.MC_AddAxisToGroup;
	{attribute 'hide'}
	fbRemoveAxisToGroup : Tc3_McCoordinatedMotion.MC_RemoveAxisFromGroup;
	{attribute 'hide'}
	fbGroupEnable 		: Tc3_McCoordinatedMotion.MC_GroupEnable;
	{attribute 'hide'}
	fbGroupDisable 		: Tc3_McCoordinatedMotion.MC_GroupDisable;
	{attribute 'hide'}
	fbGroupReadStatus 	: Tc3_McCoordinatedMotion.MC_GroupReadStatus;	
	{attribute 'hide'}
	fbUngroupAllAxes 	: Tc3_McCoordinatedMotion.MC_UngroupAllAxes;	
	{attribute 'hide'}
	fbGroupReset	 	: Tc3_McCoordinatedMotion.MC_GroupReset;
	{attribute 'hide'}
	nState_SEQ_Adding 	: UDINT;
	{attribute 'hide'}	
	fbMovers : CHALET_BaseComponents.FB_CH_List; // List of Axis to be added to the group
		
	//Link to CA Group
	GroupRef : AXES_GROUP_REF;
	
	{attribute 'hide'}	
	ipTempMover : I_XTS_Mover;

	{attribute 'hide'}
	dummyAxis : AXIS_REF;
	
	{attribute 'hide'}	
	fbFeedback : CHALET_BaseComponents.FB_CH_Feedback(ipSourceInfo := fbSourceInfo);
	
	{attribute 'hide'}
	eActiveCommand : E_NcGroupCommands := E_NcGroupCommands.None;

END_VAR

METHOD AddAxisListToGroup : HRESULT
VAR_INPUT
	ipMovers : CHALET_BaseComponents.I_CH_List;
END_VAR
IF NOT THIS^.fbFeedback.Done THEN
	//Errror active/not ready
	THIS^.fbFeedback.LastCommandAccepted := FALSE;
	
ELSIF nState_SEQ_Adding <> 0 AND nState_SEQ_Adding <> 999 THEN
	// Adding Sequence is not finished. Terminate first
	THIS^.fbFeedback.LastCommandAccepted := FALSE;

ELSIF ipMovers = 0 THEN
	// Invalide input
	THIS^.fbFeedback.LastCommandAccepted := FALSE;
		
ELSE
	// duplicate List
	THIS^.fbMovers.Duplicate(ipListCopyFrom := ipMovers);
	
	
	THIS^.nState_SEQ_Adding := 1;
	THIS^.fbFeedback.LastCommandAccepted := TRUE;
	THIS^.eActiveCommand := E_NcGroupCommands.AddAxisListToGroup;
	THIS^.fbFeedback.Busy := TRUE;	

END_IF

IF THIS^.fbFeedback.LastCommandAccepted THEN
	AddAxisListToGroup := S_OK;
ELSE
	AddAxisListToGroup := E_FAIL;
END_IF
END_METHOD

METHOD AddingAxisToGroup : HRESULT
VAR
	hr : HRESULT;
END_VAR
VAR_INST
	ipMover : CHALET_BaseComponents.I_CH_Object;
END_VAR
AddingAxisToGroup := S_PENDING;

CASE nState_SEQ_Adding OF
	0: // Idle
		AddingAxisToGroup := S_OK;
		
		
	1: // prepare List for iteratrion 
		THIS^.fbMovers.ResetIterator();
		nState_SEQ_Adding := 10;
		
		
	10: // has next Mover?
		IF THIS^.fbMovers.HasNextObject() THEN
			ipMover := THIS^.fbMovers.GetNextObject();
			IF ToMover(ipMover, ipTempMover) THEN
				nState_SEQ_Adding := 20;
			END_IF
		ELSE 
			nState_SEQ_Adding := 100;			
		END_IF
		
		
	20: // get Axis Reference
		IF ipTempMover <> 0 AND_THEN __ISVALIDREF(ipTempMover.getAxisRef) THEN
			nState_SEQ_Adding := 30;
		ELSE
			nState_SEQ_Adding := 1000 + nState_SEQ_Adding;	
		END_IF
		
		
	30: // add mover to group
		fbAddAxisToGroup.Execute := TRUE;
		IF fbAddAxisToGroup.Error THEN
			nState_SEQ_Adding := 1000 + nState_SEQ_Adding;
		ELSIF fbAddAxisToGroup.Done THEN
			nState_SEQ_Adding := 40;
			ipTempMover.MoverInGroup := TRUE;
		END_IF

	40: // Remove Object from List
		IF THIS^.fbMovers.RemoveObject(ipMover) THEN
			THIS^.fbMovers.ResetIterator();
			nState_SEQ_Adding := 10;
		ELSE
			nState_SEQ_Adding := 1000 + nState_SEQ_Adding;	
		END_IF
			
		
	100: // clear list
		// todo THIS^.iMovers.Clear();	
		nState_SEQ_Adding := 999;
		
		
	999: // Done
		AddingAxisToGroup := S_OK;

		
	1000..1999://Error
		hr := GetMostSignificant(hr, E_FAIL);	
			
END_CASE

// Propagate error
IF FAILED(hr) THEN
	AddingAxisToGroup := hr;
END_IF

// set feedback
THIS^.fbFeedback.HR := hr;
END_METHOD

PROPERTY AllAxesStanding : BOOL
GET
AllAxesStanding := fbGroupReadStatus.AllAxesStanding;
END_GET
END_PROPERTY

METHOD ChangeGapMode : HRESULT
VAR_INPUT
	bFast : BOOL;
END_VAR
ChangeGapMode := S_PENDING;

IF bFast THEN
	// Change fist to positive direction and then to Fast Mode	
	ipUtilityCAGroup.SetGapControlDirection(MC_GAP_CONTROL_DIRECTION.mcGapCtrlDirectionPositive);
	ipUtilityCAGroup.SetDefaultGapControlMode(MC_DEFAULT_GAP_CONTROL_MODE.mcGapCtrlModeFast);
ELSE
	// Change first to StandardMode and then to both direction
	ipUtilityCAGroup.SetDefaultGapControlMode(MC_DEFAULT_GAP_CONTROL_MODE.mcGapCtrlModeStandard);
	ipUtilityCAGroup.SetGapControlDirection(MC_GAP_CONTROL_DIRECTION.mcGapCtrlDirectionBoth);
END_IF

ChangeGapMode := S_OK;
END_METHOD

METHOD Disable : HRESULT
THIS^.fbFeedback.LastCommandAccepted := TRUE;
THIS^.fbFeedback.Busy := TRUE;	
THIS^.fbGroupDisable.Execute := TRUE;
THIS^.eActiveCommand := E_NcGroupCommands.GroupDisable;



IF THIS^.fbFeedback.LastCommandAccepted THEN
	Disable := S_OK;
ELSE
	Disable := E_FAIL;
END_IF
END_METHOD

METHOD Enable : HRESULT
IF NOT THIS^.fbFeedback.Done THEN
	THIS^.fbFeedback.LastCommandAccepted := FALSE;
	// Error active/not ready
	
ELSIF NOT(THIS^.fbGroupReadStatus.GroupDisabled) THEN
	THIS^.fbFeedback.LastCommandAccepted := FALSE;
	// Group in wrong State
	
ELSE
	THIS^.fbFeedback.LastCommandAccepted := TRUE;
	THIS^.fbFeedback.Busy := TRUE;
	THIS^.eActiveCommand := E_NcGroupCommands.GroupEnable;
	THIS^.fbGroupEnable.Execute := TRUE;
END_IF

IF THIS^.fbFeedback.LastCommandAccepted THEN
	Enable := S_OK;
ELSE
	Enable := E_FAIL;
END_IF
END_METHOD

METHOD FB_init : BOOL
VAR_INPUT
	bInitRetains : BOOL; // if TRUE, the retain variables are initialized (warm start / cold start)
	bInCopyCode : BOOL;  // if TRUE, the instance afterwards gets moved into the copy code (online change)
	
	ipXtsSystem : I_XTS_System_Registration; //Interface to XTS system object	
END_VAR
VAR_INST
	{attribute 'hide'}
	bFBInitCalledOnce : BOOL; //Do the following code once during start up and not during onlinechange
END_VAR
//Do the following code once during start up and not during onlinechange
IF NOT bFBInitCalledOnce THEN 
	
	//Regristrate object in System
	IF ipXtsSystem <> 0 THEN
		ipXtsSystem.LinkGroup(THIS^);
		THIS^.ipXtsSystem := ipXtsSystem;
	END_IF

END_IF

bFBInitCalledOnce := TRUE;
END_METHOD

{attribute 'monitoring':='call'}
PROPERTY GroupEnabled : BOOL
GET
GroupEnabled := fbGroupReadStatus.Valid AND NOT (fbGroupReadStatus.GroupDisabled OR fbGroupReadStatus.GroupErrorStop);
END_GET
END_PROPERTY

{attribute 'monitoring':='call'}
PROPERTY HR : HRESULT
GET
HR := fbFeedback.hr;
END_GET
END_PROPERTY

METHOD Initialize : HRESULT
VAR
	stVarInfo : __SYSTEM.VAR_INFO;
END_VAR
VAR_INST
	//This error cannot be reset. Requires a reset cold
	{attribute 'hide'}	
	fbInitError : FB_TcAlarm;
END_VAR
IF NOT THIS^.bInitDone THEN

	Initialize := S_PENDING;

	
	// Check if link to Group is mapped
	IF NcParameterlist.ERROR_IF_NC_AXIS_IS_NOT_MAPPED AND_THEN F_GetMappingStatus(ADR(THIS^.GroupRef.NcToPlc), SIZEOF(THIS^.GroupRef.NcToPlc)) <> EPlcMappingStatus.MS_Mapped THEN
		IF NOT fbInitError.bRaised THEN 
			//This error cannot be reset. Requires a reset cold
			fbInitError.CreateEx(stEventEntry := TC_EVENTS.CHALET_NC_Events.VariableLinkMissing, ipSourceInfo := THIS^.fbSourceInfo, bWithConfirmation := FALSE);
			stVarInfo := __VARINFO(GroupRef.NcToPlc);
			fbInitError.ipArguments.AddString(stVarInfo.Symbol);
			fbInitError.Raise(0);
		END_IF
		Initialize := E_FAIL;
		RETURN;
	END_IF
	
	
	// Check if link to Group is mapped
	IF NcParameterlist.ERROR_IF_NC_AXIS_IS_NOT_MAPPED AND_THEN F_GetMappingStatus(ADR(THIS^.GroupRef.PlcToNc), SIZEOF(THIS^.GroupRef.PlcToNc)) <> EPlcMappingStatus.MS_Mapped THEN
		IF NOT fbInitError.bRaised THEN 
			//This error cannot be reset. Requires a reset cold
			fbInitError.CreateEx(stEventEntry:= TC_EVENTS.CHALET_NC_Events.VariableLinkMissing, ipSourceInfo := THIS^.fbSourceInfo, bWithConfirmation := FALSE);
			stVarInfo := __VARINFO(GroupRef.PlcToNc);
			fbInitError.ipArguments.AddString(stVarInfo.Symbol);
			fbInitError.Raise(0);
		END_IF
		Initialize := E_FAIL;		
		RETURN;
	END_IF	


		
	IF THIS^.ipXtsSystem.Environment <> 0 THEN
		ipUtilityCAGroup := THIS^.ipXtsSystem.Environment.UtilityEnvirement.Mc2CaGroup(1);
	END_IF

	THIS^.bInitDone := TRUE;
ELSE
	
	Initialize := S_OK;

END_IF
END_METHOD

{attribute 'monitoring':='call'}
PROPERTY Mapped : BOOL //Project is mapped to NC (NcToPlc and PlcToNc)
GET
VAR
	bNcToPlcNotMapped 	: BOOL;
	bPlcToNcNotMapped 	: BOOL;
END_VAR
bNcToPlcNotMapped := F_GetMappingStatus(ADR(THIS^.GroupRef.NcToPlc), SIZEOF(THIS^.GroupRef.NcToPlc)) <> EPlcMappingStatus.MS_Mapped;
bPlcToNcNotMapped := F_GetMappingStatus(ADR(THIS^.GroupRef.PlcToNc), SIZEOF(THIS^.GroupRef.PlcToNc)) <> EPlcMappingStatus.MS_Mapped;

Mapped := NOT bNcToPlcNotMapped AND NOT bPlcToNcNotMapped;
END_GET
END_PROPERTY

{attribute 'monitoring':='call'}
PROPERTY OID : OTCID
GET
OID := GroupRef.NcToPlc.Common.GroupOID;
END_GET
END_PROPERTY

METHOD RemoveAxisFromGroup : HRESULT
VAR_INPUT
	ipMover	: I_XTS_Mover;
END_VAR
IF ipMover = 0 THEN
	THIS^.fbFeedback.LastCommandAccepted	:= FALSE;
	//Error no valid input
	
ELSE
	THIS^.eActiveCommand := E_NcGroupCommands.RemoveAxisFromGroup;
	THIS^.fbFeedback.LastCommandAccepted := TRUE;
	THIS^.fbFeedback.Busy := TRUE;

	fbRemoveAxisToGroup.IdentInGroup := ipMover.IdentInGroup;
	fbRemoveAxisToGroup.Execute := TRUE;
	ipMover.MoverInGroup := FALSE;
END_IF

IF THIS^.fbFeedback.LastCommandAccepted THEN
	RemoveAxisFromGroup := S_OK;
ELSE
	RemoveAxisFromGroup := E_FAIL;
END_IF
END_METHOD

METHOD Reset : HRESULT
THIS^.eActiveCommand := E_NcGroupCommands.GroupReset;
THIS^.fbFeedback.LastCommandAccepted := TRUE;
THIS^.fbFeedback.Busy := TRUE;	

THIS^.fbGroupReset.Execute := TRUE;

IF THIS^.fbFeedback.LastCommandAccepted THEN
	Reset := S_OK;
ELSE
	Reset := E_FAIL;
END_IF
END_METHOD

METHOD UngroupAllAxes : HRESULT
THIS^.eActiveCommand := E_NcGroupCommands.UngroupAllAxes;
THIS^.fbFeedback.LastCommandAccepted := TRUE;
THIS^.fbFeedback.Busy := TRUE;	

THIS^.nState_SEQ_Adding := 0;

THIS^.fbUngroupAllAxes.Execute := TRUE;


IF THIS^.fbFeedback.LastCommandAccepted THEN
	UngroupAllAxes := S_OK;
ELSE
	UngroupAllAxes := E_FAIL;
END_IF
END_METHOD

METHOD Update : HRESULT
// ********************** Refresh Group Information ***********************************************
fbGroupReadStatus(AxesGroup:=  THIS^.GroupRef, Enable:= TRUE);

// ********************** Set feedback depending on active command *******************************
IF THIS^.eActiveCommand <> E_NcGroupCommands.None THEN
	fbFeedback.ActiveCommand 	:= TO_STRING(THIS^.eActiveCommand);	
END_IF

CASE THIS^.eActiveCommand OF 
  E_NcGroupCommands.GroupDisable:
		fbFeedback.Busy 		:= fbGroupDisable.Busy;
		fbFeedback.Done 		:= fbGroupDisable.Done;
		fbFeedback.ErrorId 		:= fbGroupDisable.ErrorId;
  
  E_NcGroupCommands.GroupEnable:
		fbFeedback.Busy 		:= fbGroupEnable.Busy;
		fbFeedback.Done 		:= fbGroupEnable.Done;
		fbFeedback.ErrorId 		:= fbGroupEnable.ErrorId;
  
  E_NcGroupCommands.GroupReset:
		fbFeedback.Busy 		:= fbGroupReset.Busy;
		fbFeedback.Done 		:= fbGroupReset.Done;
		fbFeedback.ErrorId 		:= fbGroupReset.ErrorId;  
  
  E_NcGroupCommands.AddAxisListToGroup: 
		fbFeedback.Busy 		:= nState_SEQ_Adding > 0 AND nState_SEQ_Adding < 999;
		fbFeedback.Done 		:= nState_SEQ_Adding = 999; 
//		fbFeedback.ErrorId 		:= ;
  
  E_NcGroupCommands.RemoveAxisFromGroup:
		fbFeedback.Busy 		:= fbRemoveAxisToGroup.Busy;
		fbFeedback.Done 		:= fbRemoveAxisToGroup.Done;
		fbFeedback.ErrorId 		:= fbRemoveAxisToGroup.ErrorId;
  
  E_NcGroupCommands.UngroupAllAxes:
		fbFeedback.Busy 		:= fbUngroupAllAxes.Busy;
		fbFeedback.Done 		:= fbUngroupAllAxes.Done;
		fbFeedback.ErrorId 		:= fbUngroupAllAxes.ErrorId;
  
END_CASE

// **********************  Stop to execute commands on .done or .error ***************************
IF THIS^.fbFeedback.Done OR THIS^.fbFeedback.Error THEN
	THIS^.eActiveCommand 				:= E_NcGroupCommands.None;
END_IF


// **********************  Cyclic calls  *********************************************************
IF THIS^.ipTempMover <> 0 THEN
	fbAddAxisToGroup(AxesGroup := THIS^.GroupRef, Axis := THIS^.ipTempMover.getAxisRef, IdentInGroup := ipTempMover.IdentInGroup);
ELSE
	fbAddAxisToGroup(AxesGroup := THIS^.GroupRef, Axis := dummyAxis);
END_IF

fbRemoveAxisToGroup(AxesGroup := THIS^.GroupRef);
fbGroupEnable(AxesGroup := THIS^.GroupRef);
fbGroupDisable(AxesGroup := THIS^.GroupRef);
fbUngroupAllAxes(AxesGroup := THIS^.GroupRef);
fbGroupReset(AxesGroup := THIS^.GroupRef);

// ********************** Reset all Execution flags **********************************************
fbAddAxisToGroup.Execute := FALSE;
fbRemoveAxisToGroup.Execute := FALSE;
fbGroupEnable.Execute := FALSE;
fbGroupDisable.Execute := FALSE;
fbUngroupAllAxes.Execute := FALSE;
fbGroupReset.Execute := FALSE;


// todo hresult
END_METHOD

{attribute 'monitoring':='call'}
PROPERTY UtilityCAGroup : I_Mc2CaGroup
GET
UtilityCAGroup := THIS^.ipUtilityCAGroup;
END_GET
END_PROPERTY

END_FUNCTION_BLOCK

// ---- COMPENENTs/Mover/FB_XTS_Axis.TcPOU
{attribute 'no_explicit_call' := 'Do not call the body - Stick to OOP'}
FUNCTION_BLOCK FB_XTS_Axis EXTENDS CHALET_NC.FB_NcAxis IMPLEMENTS I_XTS_Axis
VAR
	{attribute 'hide'}
	fbMoveAbsoluteCA		: ARRAY [0..1] OF MC_MoveAbsoluteCA;//A second function block is always required to use the BufferMode. It is not possible to trigger a move function block with new parameters while it is active.
	{attribute 'hide'}
	fbHaltCA				: MC_HaltCA;
	{attribute 'hide'}
	nActiveMoveAbsCa 		: UINT;
END_VAR

METHOD HaltCA : I_CH_Feedback
VAR_INPUT
	fDeceleration          : LREAL;
    fJerk                  : LREAL;
    fGap                   : LREAL;
END_VAR
IF THIS^.Feedback.Error THEN
	THIS^.fbFeedback.LastCommandAccepted	:= FALSE;
	//Error active/not ready
		
ELSE
	THIS^.eActiveCommand 					:= CHALET_Nc.E_NcAxisCommands.HaltCA;
	THIS^.fbFeedback.LastCommandAccepted	:= TRUE;		
	THIS^.fbFeedback.Busy 					:= TRUE;
	                                    	
	THIS^.fbHaltCA.Execute					:= TRUE;
	THIS^.fbHaltCA.Gap						:= fGap;
	
	
	//Deceleration
	//If input = 0  then use default dynamics
	IF fDeceleration = 0.0 THEN
		THIS^.fbHaltCA.Deceleration := THIS^.fDefaultDeceleration;
	ELSE
		THIS^.fbHaltCA.Deceleration := fDeceleration;
	END_IF
	
	//Jerk
	//If input = 0  then use default dynamics
	IF fJerk = 0.0 THEN
		THIS^.fbHaltCA.Jerk := THIS^.fDefaultJerk;
	ELSE
		THIS^.fbHaltCA.Jerk := fJerk;
	END_IF

END_IF


HaltCA := THIS^.fbFeedback;
END_METHOD

{attribute 'TcRpcEnable':='1'} //call methode via OPC-UA conection
METHOD MoveAbsoluteCA  : I_CH_Feedback
VAR_INPUT
	fPosition		: LREAL;
	
	(* This value determines the minimum gap to the predecessor for Collision Avoidance. *)
	fGap			: LREAL;
	
	(* Use the default dynamics if input=0. 
	The default dynamics can be read and written via property and is initialized with the default values in the NC parameter list. *)
	fVelocity		: LREAL;
	
	(* Use the default dynamics if input=0. 
	The default dynamics can be read and written via property and is initialized with the default values in the NC parameter list. *)
	fAcceleration	: LREAL;
	
	(* Use the default dynamics if input=0. 
	The default dynamics can be read and written via property and is initialized with the default values in the NC parameter list. *)
	fDeceleration	: LREAL;
	
	(* Use the default dynamics if input=0. 
	The default dynamics can be read and written via property and is initialized with the default values in the NC parameter list. *)
	fJerk			: LREAL;
	
	(* Defines the direction of the movement (e.g. for a modulo axis). 
		input=0 = mcDirectionNonModulo*)
	eDirection	: Tc3_Mc3Definitions.MC_DIRECTION;
	
	(* Use the Aborting mode without buffering if input=0. 
	BufferModes:
		-MC_Aborting: Default mode without buffering. The command is executed immediately and interrupts any other command that may be running.
		-MC_Buffered: The command is executed once no other command is running on the axis. The previous movement continues until it has stopped. The following command is started from standstill. *)
	eBufferMode   : Tc3_Mc3Definitions.MC_BUFFER_MODE;
END_VAR
VAR
	nInactiveInstance : UINT;
END_VAR
IF THIS^.Feedback.Error THEN
	THIS^.fbFeedback.LastCommandAccepted	:= FALSE;
	//Error active/not ready

ELSIF NOT THIS^.BufferEmpty THEN		
	THIS^.fbFeedback.LastCommandAccepted	:= FALSE;
	//Buffer not ready to store next motion command	
	
ELSIF NOT((eBufferMode <> Tc3_Mc3Definitions.MC_BUFFER_MODE.mcAborting) OR (eBufferMode <> Tc3_Mc3Definitions.MC_BUFFER_MODE.mcBuffered)) THEN		
	THIS^.fbFeedback.LastCommandAccepted	:= FALSE;
	//only mcAborting and mcBuffered are available 	
	
ELSIF NOT(THIS^.Axis.Status.StandStill OR THIS^.Axis.Status.DiscreteMotion OR THIS^.Axis.Status.ContinuousMotion OR THIS^.Axis.Status.SynchronizedMotion) THEN		
	THIS^.fbFeedback.LastCommandAccepted	:= FALSE;
	//Axis in wrong State
	
ELSIF (eBufferMode <> Tc3_Mc3Definitions.MC_BUFFER_MODE.mcAborting) AND bNewBufferCommadThisCycle THEN		
	THIS^.fbFeedback.LastCommandAccepted	:= FALSE;
	//Buffer not ready to store next motion command		
	//Max send one buffered motion command each cycle	
	
ELSE
	//A second function block is always required to use the BufferMode. It is not possible to trigger a move function block with new parameters while it is active.
	IF THIS^.fbMoveAbsoluteCA[nActiveMoveAbsCA].Busy THEN
		nInactiveInstance := (THIS^.nActiveMoveAbsCa + 1)MOD 2;
	ELSE
		nInactiveInstance := THIS^.nActiveMoveAbsCa;
	END_IF
	
	THIS^.eActiveCommand 				:= E_NcAxisCommands.MoveAbsoluteCA;
	THIS^.fbFeedback.LastCommandAccepted:= TRUE;		
	THIS^.fbFeedback.Busy 				:= TRUE;
	
	THIS^.fbMoveAbsoluteCA[nInactiveInstance].ContinuousUpdate := TRUE;
	THIS^.fbMoveAbsoluteCA[nInactiveInstance].Execute		:= TRUE;
	THIS^.fbMoveAbsoluteCA[nInactiveInstance].Gap			:= fGap;
	THIS^.fbMoveAbsoluteCA[nInactiveInstance].Position		:= fPosition;
	THIS^.fbMoveAbsoluteCA[nInactiveInstance].Direction		:= eDirection;
	THIS^.fbMoveAbsoluteCA[nInactiveInstance].BufferMode 	:= eBufferMode;
	
	//If the currend command is a buffered movement, then set a flag.
	IF eBufferMode <> Tc3_Mc3Definitions.MC_BUFFER_MODE.mcAborting THEN
		THIS^.bNewBufferCommadThisCycle := TRUE;
	END_IF
	
	//Velocity
	//If input = 0  then use default dynamics
	IF fVelocity = 0.0 THEN
		THIS^.fbMoveAbsoluteCA[nInactiveInstance].Velocity := THIS^.fDefaultVelocity;
	ELSE
		THIS^.fbMoveAbsoluteCA[nInactiveInstance].Velocity := fVelocity;
	END_IF
	
	//Acceleration
	//If input = 0  then use default dynamics
	IF fAcceleration = 0.0 THEN
		THIS^.fbMoveAbsoluteCA[nInactiveInstance].Acceleration := THIS^.fDefaultAcceleration;
	ELSE
		THIS^.fbMoveAbsoluteCA[nInactiveInstance].Acceleration := fAcceleration;
	END_IF
	
	//Deceleration
	//If input = 0  then use default dynamics
	IF fDeceleration = 0.0 THEN
		THIS^.fbMoveAbsoluteCA[nInactiveInstance].Deceleration := THIS^.fDefaultDeceleration;
	ELSE
		THIS^.fbMoveAbsoluteCA[nInactiveInstance].Deceleration := fDeceleration;
	END_IF
	
	//Jerk
	//If input = 0  then use default dynamics
	IF fJerk = 0.0 THEN
		THIS^.fbMoveAbsoluteCA[nInactiveInstance].Jerk := THIS^.fDefaultJerk;
	ELSE
		THIS^.fbMoveAbsoluteCA[nInactiveInstance].Jerk := fJerk;
	END_IF

END_IF


MoveAbsoluteCA := THIS^.fbFeedback;
END_METHOD

METHOD Update  : HRESULT
// ********************** Do initialisation first ***********************************************
IF NOT bInitDone THEN
	Update := THIS^.Initialize();
	RETURN;
END_IF

// ********************** Set feedback depending on active command *******************************
CASE THIS^.eActiveCommand OF                                                                      
	E_NcAxisCommands.MoveAbsoluteCA:                                                              
		fbFeedback.Busy 		:= fbMoveAbsoluteCA[nActiveMoveAbsCa].Busy;                       
		fbFeedback.Done 		:= fbMoveAbsoluteCA[nActiveMoveAbsCa].Done;                       
		fbFeedback.ErrorId 		:= fbMoveAbsoluteCA[nActiveMoveAbsCa].ErrorID;  
       
	E_NcAxisCommands.HaltCA:                                                              
		fbFeedback.Busy 		:= fbHaltCA.Busy;                       
		fbFeedback.Done 		:= fbHaltCA.Done OR fbHaltCA.CommandAborted;                       
		fbFeedback.ErrorId 		:= fbHaltCA.ErrorID;            
END_CASE                                                                                          

// **********************  Cyclic call super Update  *********************************************
SUPER^.Update();
                                                                                                  
                                                                                                  
// **********************  Cyclic calls  *********************************************************
fbMoveAbsoluteCA[0](Axis := THIS^.Axis);                                                          
fbMoveAbsoluteCA[1](Axis := THIS^.Axis);                                                          
fbHaltCA(Axis := THIS^.Axis);
                                                                                                
                                                                                                  
// ********************** Reset all Execution flags **********************************************
fbMoveAbsoluteCA[0].Execute := FALSE;                                                             
fbMoveAbsoluteCA[1].Execute := FALSE;
fbHaltCA.Execute := FALSE;                                                                                                  

                                                                                                 
// ****************Get the acive instance. Stay at the last active.*******************************
IF fbMoveAbsoluteCA[0].Active THEN                                                                
	nActiveMoveAbsCa := 0;
ELSIF fbMoveAbsoluteCA[1].Active THEN
	nActiveMoveAbsCa := 1;
END_IF

//Return
Update := THIS^.fbFeedback.HR;
END_METHOD

END_FUNCTION_BLOCK

// ---- COMPENENTs/Mover/FB_XTS_Mover.TcPOU
{attribute 'no_explicit_call' := 'Do not call the body - Stick to OOP'}
FUNCTION_BLOCK FB_XTS_Mover EXTENDS FB_CH_Object IMPLEMENTS I_XTS_Mover, I_XTS_Mover_PLC
VAR	
	//Link to NC
	Axis : FB_XTS_Axis;

	{attribute 'hide'}
	bInitDone : BOOL;
	{attribute 'hide'}
	ipXtsSystem : I_XTS_System_Registration;
	{attribute 'hide'}
	ipUtilityMover : I_TcIoXtsXpuMover;
	{attribute 'hide'}
	ipProductData : I_XTS_ProductData; //later the required interface of the tool or product can be queried via query interface
	{attribute 'hide'}
	ipParentStation : I_XTS_Station; //This is the station in which the Mover is currently standing or moving.	
	{attribute 'hide'}
	ipNextMover : I_XTS_Mover;
	{attribute 'hide'}
	sTargedStation : STRING;
	{attribute 'hide'}
	fLastCmdTargedPosition : LREAL; //the last commanded target position [mm]
	{attribute 'hide'}
	fLastCmdTargedVelocity : LREAL; //the last commanded target speed
	{attribute 'hide'}	
	fLastCmdTargedGap 	: LREAL; //the last commanded target gap
	{attribute 'hide'}
	bInGroup : BOOL;	
	{attribute 'hide'}	
	lrTrackLentgh 			: LREAL; //[mm]  Modulo
	{attribute 'hide'}
	fbFeedback 					: CHALET_BaseComponents.FB_CH_Feedback(ipSourceInfo := fbSourceInfo);;
	
END_VAR
VAR PERSISTENT
	fDrivenDistance : LREAL;
END_VAR

{attribute 'monitoring':='call'}
PROPERTY Coupled : BOOL
GET
Coupled := THIS^.Axis.Coupled;
END_GET
END_PROPERTY

{attribute 'OPC.UA.DA.Property' := '1'}
{attribute 'monitoring':='call'}
PROPERTY DefaultAcceleration : LREAL
GET
DefaultAcceleration := THIS^.Axis.DefaultAcceleration;
END_GET
SET
THIS^.Axis.DefaultAcceleration := DefaultAcceleration;
END_SET
END_PROPERTY

{attribute 'OPC.UA.DA.Property' := '1'}
{attribute 'monitoring':='call'}
PROPERTY DefaultDeceleration : LREAL
GET
DefaultDeceleration := THIS^.Axis.DefaultDeceleration;
END_GET
SET
THIS^.Axis.DefaultDeceleration := DefaultDeceleration;
END_SET
END_PROPERTY

{attribute 'OPC.UA.DA.Property' := '1'}
{attribute 'monitoring':='call'}
PROPERTY DefaultJerk : LREAL
GET
DefaultJerk := THIS^.Axis.DefaultJerk;
END_GET
SET
THIS^.Axis.DefaultJerk := DefaultJerk;
END_SET
END_PROPERTY

METHOD Disable : HRESULT
Axis.PowerOff();


//Show as feedback the state of the includet axis
fbFeedback.ActiveCommand := Axis.Feedback.ActiveCommand;
fbFeedback.LastCommandAccepted := Axis.Feedback.LastCommandAccepted;
fbFeedback.HR := Axis.Feedback.hr;


IF Axis.Feedback.LastCommandAccepted THEN
	Disable := S_OK;
ELSE  
	Disable := E_FAIL;;	
END_IF
END_METHOD

{attribute 'monitoring':='call'}
PROPERTY DrivenDistance : LREAL
GET
DrivenDistance := fDrivenDistance;
END_GET
END_PROPERTY

METHOD Enable : HRESULT
Axis.PowerOn();


//Show as feedback the state of the includet axis
fbFeedback.ActiveCommand := Axis.Feedback.ActiveCommand;
fbFeedback.LastCommandAccepted := Axis.Feedback.LastCommandAccepted;
fbFeedback.HR := Axis.Feedback.hr;


IF Axis.Feedback.LastCommandAccepted THEN
	Enable := S_OK;
ELSE  
	Enable := E_FAIL;;	
END_IF
END_METHOD

METHOD FB_init : BOOL
VAR_INPUT
	bInitRetains : BOOL; // if TRUE, the retain variables are initialized (warm start / cold start)
	bInCopyCode : BOOL;  // if TRUE, the instance afterwards gets moved into the copy code (online change)
	
	ipXtsSystem : I_XTS_System_Registration; //Interface to XTS system object
END_VAR
VAR_INST
	{attribute 'hide'}
	bFBInitCalledOnce : BOOL; //Do the following code once during start up and not during onlinechange
END_VAR
//Do the following code once during start up and not during onlinechange
IF NOT bFBInitCalledOnce THEN 
	

	//Regristrate object in System
	IF ipXtsSystem <> 0 THEN
		ipXtsSystem.RegisterMover(THIS^);
		THIS^.ipXtsSystem := ipXtsSystem;
	END_IF


	
END_IF

bFBInitCalledOnce := TRUE;
END_METHOD

{attribute 'monitoring':='call'}
PROPERTY Feedback : I_CH_Feedback
GET
Feedback := THIS^.fbFeedback;
END_GET
END_PROPERTY

(*The _ PLC interface provides the user with a simplified interface for commanding between the stations. Sometimes, however, this is not enough. 
Either you get the corresponding interface with the __Queryinterface or you can get full access with this property.*)
PROPERTY FullAccess : I_XTS_Mover
GET
FullAccess := (THIS^);
END_GET
END_PROPERTY

PROPERTY getAxisRef : REFERENCE TO Tc2_MC2.AXIS_REF
GET
getAxisRef REF= THIS^.Axis.getAxisRef;
END_GET
END_PROPERTY

METHOD HaltCA : HRESULT
VAR_INPUT
END_VAR
Axis.HaltCA(
	fDeceleration:= 0, //use default
	fJerk:= 0, //use default
	fGap:= fLastCmdTargedGap);
	

//Show as feedback the state of the includet axis
fbFeedback.ActiveCommand := Axis.Feedback.ActiveCommand;
fbFeedback.LastCommandAccepted := Axis.Feedback.LastCommandAccepted;
fbFeedback.HR := Axis.Feedback.hr;


IF Axis.Feedback.LastCommandAccepted THEN
	HaltCA := S_OK;
ELSE  
	HaltCA := E_FAIL;;	
END_IF
END_METHOD

PROPERTY IdentInGroup : IDENT_IN_GROUP_REF
GET
IdentInGroup := UDINT_TO_IDENTINGROUP(THIS^.Axis.getAxisRef.NcToPlc.AxisId);
END_GET
END_PROPERTY

METHOD Initialize : HRESULT
VAR

END_VAR

IF NOT THIS^.bInitDone THEN
	THIS^.fbFeedback.ActiveCommand 		:= TO_STRING(E_NcAxisCommands.Initialize);
	//THIS^.eActiveCommand 				:= E_NcAxisCommands.Initialize;
	THIS^.fbFeedback.LastCommandAccepted:= TRUE;		

	
	//Get Tracklength from system
	THIS^.lrTrackLentgh := THIS^.ipXtsSystem.TrackLength;
	
	
	//Validate Settings
	IF (lrTrackLentgh <= 0) THEN
		Initialize := GetMostSignificant(Initialize, E_FAIL);		
	END_IF
	

	//If only one mover is in project, then interface stays 0.
	IF THIS^.ipXtsSystem.Movers.Size > 1 THEN
		THIS^.ipNextMover := THIS^.ipXtsSystem.getMoverInFront(THIS^);
		//Validate Settings
		IF (ipNextMover = 0) THEN
			Initialize := GetMostSignificant(Initialize, E_FAIL);	
		END_IF
	ELSE
		THIS^.ipNextMover := 0;
	END_IF
	
	// Get XTS Utility mover object
	IF ipXtsSystem.Environment <> 0 THEN
		ipUtilityMover := ipXtsSystem.Environment.UtilityEnvirement.GetMoverInterfaceByAxisId(THIS^.getAxisRef.NcToPlc.AxisId);
		//Validate 
		IF (ipUtilityMover = 0) THEN
			Initialize := GetMostSignificant(Initialize, E_FAIL);	
		END_IF
	END_IF
	
	
	//InitAxis
	Initialize := GetMostSignificant(Initialize, Axis.Initialize());	

	bInitDone := CheckOk(Initialize);
END_IF

fbFeedback.hr := Initialize;;
END_METHOD

{attribute 'monitoring':='call'}
PROPERTY LagDistance : LREAL
GET
LagDistance := THIS^.Axis.LagDistance;
END_GET
END_PROPERTY

{attribute 'monitoring':='call'}
PROPERTY LastCmdTargedGap : LREAL
GET
LastCmdTargedGap := fLastCmdTargedGap;
END_GET
END_PROPERTY

{attribute 'monitoring':='call'}
PROPERTY LastCmdTargedPosition : LREAL
GET
LastCmdTargedPosition := fLastCmdTargedPosition;
END_GET
END_PROPERTY

{attribute 'monitoring':='call'}
PROPERTY LastCmdTargedVelocity : LREAL
GET
LastCmdTargedVelocity := fLastCmdTargedVelocity;
END_GET
END_PROPERTY

METHOD MoveAbsCA : HRESULT
VAR_INPUT
	fPosition	: LREAL := MC_INVALID;
	fVelocity	: LREAL := MC_INVALID;
	fGap		: LREAL := MC_DEFAULT;
	eDirection	: Tc3_Mc3Definitions.MC_DIRECTION;
END_VAR
Axis.MoveAbsoluteCA(
	fPosition:= fPosition, 
	fVelocity:= fVelocity, 
	fGap:= fGap, 
	fAcceleration:= 0, //Use Axis default
	fDeceleration:= 0, //Use Axis default
	fJerk:= 0, 			//Use Axis default
	eDirection := eDirection,
	eBufferMode:= Tc3_Mc3Definitions.MC_BUFFER_MODE.mcAborting);

THIS^.fLastCmdTargedVelocity := fVelocity;
THIS^.fLastCmdTargedPosition := fPosition;
THIS^.fLastCmdTargedGap := fGap;


//Show as feedback the state of the includet axis
fbFeedback.ActiveCommand := Axis.Feedback.ActiveCommand;
fbFeedback.LastCommandAccepted := Axis.Feedback.LastCommandAccepted;
fbFeedback.HR := Axis.Feedback.hr;


IF Axis.Feedback.LastCommandAccepted THEN
	MoveAbsCA := S_OK;
ELSE  
	MoveAbsCA := E_FAIL;;	
END_IF
END_METHOD

//Returns the ID of the mover.
{attribute 'monitoring':='call'}
PROPERTY MoverID : STRING(3)
GET
IF NOT UtilityMover.P_IsInitialized THEN
	RETURN;
END_IF


MoverID := UtilityMover.GetMoverId();
END_GET
END_PROPERTY

{attribute 'monitoring':='call'}
PROPERTY MoverInGroup : BOOL
GET
MoverInGroup := bInGroup;
END_GET
SET
bInGroup := MoverInGroup;
END_SET
END_PROPERTY

{attribute 'monitoring':='call'}
PROPERTY Moving : BOOL
GET
Moving := THIS^.Axis.Moving;
END_GET
END_PROPERTY

{attribute 'monitoring':='call'}
PROPERTY NameXtsMover : STRING
GET
VAR
	ipComObject : ITComObject;
	sName : STRING;
END_VAR
IF NOT UtilityMover.P_IsInitialized THEN
	RETURN;
END_IF

///todo zzz: add oid of xts mover
FW_ObjMgr_GetObjectInstance(oid:= THIS^.UtilityMover.P_AxisOid, iid:= TC_GLOBAL_IID_LIST.IID_ITComObject, pipUnk:= ADR(ipComObject));

IF ipComObject = 0 THEN
	// Error unknown object id
	RETURN;
END_IF

ipComObject.TcGetObjectName(objName := ADR(sName), nameLen := SIZEOF(sName));


ipComObject.TcRelease();	


NameXtsMover := sName;
END_GET
END_PROPERTY

{attribute 'monitoring':='call'}
//Interface to the underlying NC axis object. Not all commands may be compatible with the CA group
PROPERTY NcAxis : I_XTS_Axis
GET
NcAxis := THIS^.Axis;
END_GET
END_PROPERTY

{attribute 'monitoring':='call'}
PROPERTY NextMover : I_XTS_Mover
GET
NextMover := ipNextMover;
END_GET
END_PROPERTY

{attribute 'monitoring':='call'}
PROPERTY OID : OTCID
GET
OID := THIS^.Axis.OID;
END_GET
END_PROPERTY

{attribute 'monitoring':='call'}
PROPERTY ParentStation : I_XTS_Station
GET
ParentStation := ipParentStation;
END_GET
SET
ipParentStation := ParentStation;
END_SET
END_PROPERTY

{attribute 'monitoring':='call'}
PROPERTY PositionOnTrack : LREAL
GET
//Round to 3 digits. If Axis is not enabled, use act position
IF THIS^.Axis.getAxisRef.Status.Disabled THEN
	PositionOnTrack := TO_LREAL(TRUNC(THIS^.Axis.ActPosModulo*1000))/1000;
ELSE
	PositionOnTrack := TO_LREAL(TRUNC(THIS^.Axis.SetPosModulo*1000))/1000;	
END_IF
END_GET
END_PROPERTY

{attribute 'monitoring':='call'}
PROPERTY PUBLIC ProductData : I_XTS_ProductData
GET
ProductData := ipProductData;
END_GET
SET
// No change. Same interface is set again
IF ipProductData = ProductData THEN
	;//Noting
	
ELSE

	// If allready an interface is linked. Unlink
	IF ipProductData <> 0 THEN
		ipProductData.LinkToMover(0);
		ipProductData := 0;
	END_IF
	
	// Link and store new interface
	IF ProductData <> 0 THEN
		ProductData.LinkToMover(THIS^);
		ipProductData := ProductData;
	END_IF
END_IF
END_SET
END_PROPERTY

METHOD Reset : HRESULT
Axis.Reset();

//Show as feedback the state of the includet axis
fbFeedback.ActiveCommand := Axis.Feedback.ActiveCommand;
fbFeedback.LastCommandAccepted := Axis.Feedback.LastCommandAccepted;
fbFeedback.HR := Axis.Feedback.hr;


IF Axis.Feedback.LastCommandAccepted THEN
	Reset := S_OK;
ELSE  
	Reset := E_FAIL;;	
END_IF
END_METHOD

{attribute 'monitoring':='call'}
PROPERTY SetAcceleration : LREAL
GET
SetAcceleration := THIS^.Axis.SetAcceleration;
END_GET
END_PROPERTY

{attribute 'monitoring':='call'}
PROPERTY SetVelocity : LREAL
GET
SetVelocity := THIS^.Axis.SetVelocity;
END_GET
END_PROPERTY

{attribute 'monitoring':='call'}
PROPERTY TargedStation : STRING
GET
TargedStation := sTargedStation;
END_GET
SET
sTargedStation := TargedStation;
END_SET
END_PROPERTY

METHOD Update : HRESULT
VAR
	fDistanceThisCycle : LREAL;
END_VAR
VAR_INST
	fLastMoverPosition : LREAL;
END_VAR
// Total distance traveled by the mover
IF Axis.Moving THEN
	fDistanceThisCycle := ABS(Axis.SetPosModulo-fLastMoverPosition);
	IF fDistanceThisCycle > (THIS^.lrTrackLentgh*0.5) THEN
		fDistanceThisCycle := THIS^.lrTrackLentgh-fDistanceThisCycle;
	END_IF
	fDrivenDistance := fDrivenDistance + fDistanceThisCycle;
END_IF

fLastMoverPosition := Axis.SetPosModulo;

Axis.Update();

//Show as feedback the state of the includet axis
fbFeedback.ActiveCommand := Axis.Feedback.ActiveCommand;
fbFeedback.HR := Axis.Feedback.hr;
END_METHOD

{attribute 'monitoring':='call'}
PROPERTY UtilityMover : I_TcIoXtsXpuMover
GET
UtilityMover := ipUtilityMover;
END_GET
END_PROPERTY

END_FUNCTION_BLOCK

// ---- COMPENENTs/Mover/ProductData/FB_XTS_ProductData.TcPOU
FUNCTION_BLOCK FB_XTS_ProductData EXTENDS FB_CH_Object IMPLEMENTS I_XTS_ProductData
VAR
	{attribute 'hide'}
	ipMover : I_XTS_Mover_PLC;
END_VAR

{attribute 'monitoring':='call'}
PROPERTY LinkedMover : I_XTS_Mover_PLC
GET
LinkedMover := ipMover;
END_GET
END_PROPERTY

METHOD LinkToMover : BOOL //it is not necessary to call this method. This is already done internally
VAR_INPUT
	ipMoverPlc : I_XTS_Mover_PLC;
END_VAR
THIS^.ipMover := ipMoverPlc;
END_METHOD

END_FUNCTION_BLOCK

// ---- COMPENENTs/Lubrication/FB_LubricationXTS.TcPOU
FUNCTION_BLOCK FB_LubricationXTS

VAR_INPUT	
	SysType:				E_SystemType;				//System type BekaPico or SkfETP2WZ
	LubMode:				E_LubricationMode;			//Lubrication Mode
	
	Execute:				BOOL;						//Triggers the function block with rising edge
	
	LubAmount:				LREAL;						//Amount of lubricant in ml/d/m/feedline(guidline is 0.21 ml at 1 m/s average velocity) or ml/100.000m/m/feedline (guidline is 0.25 ml at 1 m/s average velocity)
	
	FeedlineGap:			LREAL;						//Shortest distance between to feedlines in m (3 m is recommended max. / keep evenly spaced distances between feedlines)
	NumFeedlines:			INT;						//Number of feed lines linked to the lubrication system	(max. is 8 lines)
	OutletDosing:			LREAL;						//Amount of lubrication for single outlet in ml/round (guidline is 0.01 ml or 0.005 ml / use same outlet type for each feedline!)
END_VAR

VAR_IN_OUT
	XTSUnitRef:				I_XtsUnit//FB_XtsUnit;					//Refrence to XTSUnit
END_VAR

VAR_OUTPUT
	Busy:					BOOL;						//Shows if pumping sequence /stroke is started
	Active:					BOOL;						//Shows if function block is running
	Error:					BOOL;						//Shows if error has occured
	ErrorId:				UDINT;						//Gives respective error id
END_VAR

VAR
	//Inputs
	eSysType:				E_SystemType;
	eLubMode:				E_LubricationMode;
	bExecute:				BOOL;
	fLubAmount:				LREAL;
	fFeedlineGap:			LREAL;
	nNumFeedlines:			INT;
	fOutletDosing:			LREAL;

	//Trigger
	fbExecuteRTrig:			R_Trig;
	fbExecuteFTrig:			F_Trig;
	
	
	nFbState:				INT;
	
	nStrokesPerDay:			INT;
	tPauseTime:				TIME;
	
	fMaxDistanceDriven:		LREAL;
	fMaxDistanceDrivenTemp:	LREAL;
	fTriggerDistance:		LREAL;
	
	I:						INT;
	
	nOperationMode: 		INT;
	nRunningMode: 			INT;
	
	nNumMover:				DINT;
	nMoverIndex: 			DINT;
	
	fbTON:					TON;
	fbStrokeFTrig:			F_Trig;
	bStrokeDone:			BOOL;			
	
	ObLubOn AT %Q*:			BOOL;
	IbLubDone 	AT %I*:		BOOL;
	IbLubFull AT %I*:		BOOL;
	
	//XTS Unit
	
	
END_VAR

//ENGINEERING-SAMPLE!!!
//This FB is an engineering-sample for the control of the recommended lubrication system. Use on own risk!


//Checks if lubrication is enabled
fbExecuteRTrig(CLK:=Execute);
fbExecuteFTrig(CLK:=Execute);

//With rising edge of excecute
IF fbExecuteRTrig.Q THEN
	
	//Update intern variables
	eSysType:=SysType;
	eLubMode:=LubMode;
	
	bExecute:=Execute;
	
	fLubAmount:=LubAmount;
	
	fFeedlineGap:=FeedlineGap;
	nNumFeedlines:=NumFeedlines;
	fOutletDosing:=OutletDosing;
	
	//Switch state
	nFbState:=1;
	nOperationMode:=1;
	nRunningMode:=1;
		
	//Set status
	Active:=TRUE;

//With falling edge of execute
ELSIF fbExecuteFTrig.Q THEN
	
	//Switch state
	nFbState:=0;
	nOperationMode:=0;
	nRunningMode:=0;
	
	//Reset
	fbTon(In:=FALSE);
	fMaxDistanceDrivenTemp:=0;
	fMaxDistanceDriven:=0;
	nMoverIndex:=1;
	obLubOn:=FALSE;
	bStrokeDone:=FALSE;
	fbStrokeFTrig(Clk:=TRUE);
	
	//Set status
	Active:=FALSE;
	Busy:=FALSE;
	Error:=FALSE;
	ErrorId:=0;
END_IF


CASE nFbState OF
	0: //Idle
	
	1:	//Execute

		//Check which lubrication system is used in the application
		CASE eSysType OF
			
			0: //BekaPico
				CASE nOperationMode OF
					
					0: //Idle
						
					1: 	//Calculate data and set mode
						IF eLubMode=0 THEN
							
							IF fOutletDosing > 0 AND fLubAmount >= 0 AND fFeedlineGap > 0 THEN
								nStrokesPerDay:=LREAL_TO_INT((fLubAmount*fFeedlineGap)/fOutletDosing);
								tPauseTime:=LREAL_TO_TIME(((1000*60*60*24)-(4000*nStrokesPerDay))/nStrokesPerDay);
								
							ELSE
								Active:=FALSE;
									
								Error:=TRUE;
								ErrorId:=16#0003;
								//{error 'Wrong input values for FB'}
							
								nRunningMode:=0;
								nOperationMode:=0;
								nFbState:=0;
							END_IF
							
							nOperationMode:=2;
						
						ELSIF eLubMode=1 THEN
							
							IF fOutletDosing > 0 AND fLubAmount >= 0 AND fFeedlineGap > 0 THEN
								fTriggerDistance:=100000000*(fOutletDosing/(fLubAmount*fFeedlineGap));
								fMaxDistanceDrivenTemp:=0;

							ELSE
								Active:=FALSE;
									
								Error:=TRUE;
								ErrorId:=16#0003;
							
								nRunningMode:=0;
								nOperationMode:=0;
								nFbState:=0;
							END_IF
						
							nOperationMode:=3;
						
						ELSIF eLubMode=2 THEN
							
							nOperationMode:=4;
						ELSE
							Active:=FALSE;
									
							Error:=TRUE;
							ErrorId:=16#0003;
						
							nRunningMode:=0;
							nOperationMode:=0;
							nFbState:=0;
						END_IF
						
					
					2: //Lubrication running in time based mode
						CASE nRunningMode OF
							0: //Idle
							
							
							1: //Check if Pump is full
								IF NOT IbLubFull THEN
									Active:=FALSE;
									
									Error:=TRUE;
									ErrorId:=16#0002;
								
									nRunningMode:=0;
									nOperationMode:=0;
									nFbState:=0;	
							
								ELSE	
									nRunningMode:=2;
								END_IF
								
							2: //Pumping (1 cycle = 1 OutletDosing per Feedline)
								Busy:=TRUE;
								ObLubOn:=TRUE;
								
								fbTON(IN:=TRUE,PT:=T#5S);	
							
								IF 	fbTON.ET > T#2S  AND NOT IbLubDone  THEN
									fbTON(IN:=FALSE);
									
									ObLubOn:=FALSE;
									Busy:=FALSE;
	
									nRunningMode:=3;
									
								ELSIF (fbTon.Q AND IbLubDone) OR (fbTON.ET > T#1S AND NOT IbLubDone) THEN
									fbTON(IN:=FALSE);
									ObLubOn:=FALSE;
									
									Busy:=FALSE;
									Active:=FALSE;
									Error:=TRUE;
									ErrorId:=16#0001;
									
									nRunningMode:=0;
									nOperationMode:=0;
									nFbState:=0;		
								END_IF
						
							3: //Waiting (calculated waiting time)
								fbTON(IN:=TRUE,PT:=tPauseTime);
								
								IF fbTON.Q THEN
									fbTON(IN:=FALSE);
									
									nRunningMode:=1;
								END_IF
								
						END_CASE
	
					3: //Lubrication running in distance based mode
						
						CASE nRunningMode OF
							0: //Idle
							
							
							1: //Check if Pump is full
								IF NOT IbLubFull THEN
									Active:=FALSE;
									
									Error:=TRUE;
									ErrorId:=16#0002;
								
									nRunningMode:=0;
									nOperationMode:=0;
									nFbState:=0;	
							
								ELSE	
									nRunningMode:=2;
								END_IF
								
								
							2: //Pumping (1 cycle = 1 OutletDosing per Feedline)
								Busy:=TRUE;
								ObLubOn:=TRUE;
								
								fbTON(IN:=TRUE,PT:=T#5S);	
							
								IF 	fbTON.ET > T#1S  AND NOT IbLubDone  THEN
									fbTON(IN:=FALSE);
									
									ObLubOn:=FALSE;
									Busy:=FALSE;
	
									nRunningMode:=3;
									
								ELSIF (fbTon.Q AND IbLubDone) OR (fbTON.ET > T#1S AND NOT IbLubDone) THEN
									fbTON(IN:=FALSE);
									ObLubOn:=FALSE;
									
									Busy:=FALSE;
									Active:=FALSE;
									Error:=TRUE;
									ErrorId:=16#0001;
									
									nRunningMode:=0;
									nOperationMode:=0;
									nFbState:=0;		
								END_IF
								
								
							3: //Check how far movers have moved
								FOR nNumMover:= 1 TO XTSUnitRef.stXtsUnit.stMotion.nAxisCount DO
								
									IF XTSUnitRef.stXtsUnit.stTcIoXtsDrv.stMover[nNumMover].stParameter.fDistanceDriven > fMaxDistanceDriven THEN
										fMaxDistanceDriven:= XTSUnitRef.stXtsUnit.stTcIoXtsDrv.stMover[nNumMover].stParameter.fDistanceDriven;
										nMoverIndex:=nNumMover;
									END_IF
									
								END_FOR	
								
								fMaxDistanceDriven:=fMaxDistanceDriven-fMaxDistanceDrivenTemp;
								
								IF fMaxDistanceDriven >= fTriggerdistance THEN
									fMaxDistanceDrivenTemp:=XTSUnitRef.stXtsUnit.stTcIoXtsDrv.stMover[nMoverIndex].stParameter.fDistanceDriven;
									
									nRunningMode:=1;
								END_IF
								
						END_CASE
			
					4: //Lubrication running in continous mode
					
						CASE nRunningMode OF
							0: //Idle
						
							1: //Pumping continous
								IF NOT IbLubFull THEN
									Active:=FALSE;
									
									Error:=TRUE;
									ErrorId:=16#0002;
								
									nRunningMode:=0;
									nOperationMode:=0;
									nFbState:=0;
									
								ELSE	
									Busy:=TRUE;
									ObLubOn:=TRUE;
									
									fbTON(IN:=TRUE,PT:=T#5S);
									
									fbStrokeFTrig(Clk:=IbLubDone);
									
									IF fbStrokeFTrig.Q THEN
										bStrokeDone:=TRUE;
									END_IF
									
									IF 	fbTON.Q  AND NOT bStrokeDone THEN
										fbTON(IN:=FALSE);
										ObLubOn:=FALSE;
										
										Busy:=FALSE;
										Active:=FALSE;
										Error:=TRUE;
										ErrorId:=16#0001;
										
										nRunningMode:=0;
										nOperationMode:=0;
										nFbState:=0;
										
									ELSIF  bStrokeDone THEN
										fbTON(IN:=FALSE);
										bStrokeDone:=FALSE;
									END_IF
								
								END_IF
							
						END_CASE	
					
				END_CASE			
			
			1: //SkfETP2WZ
				CASE nOperationMode OF
					
					0: //Idle
						
					1: 	//Calculate data and set mode
						IF eLubMode=0 THEN
							
							IF fOutletDosing > 0 AND fLubAmount >= 0 AND fFeedlineGap > 0 THEN
								nStrokesPerDay:=LREAL_TO_INT((fLubAmount*fFeedlineGap)/fOutletDosing);
								tPauseTime:=LREAL_TO_TIME(((1000*60*60*24)-(420000*nStrokesPerDay))/nStrokesPerDay);
								
								IF tPauseTime < T#30M THEN
									tPauseTime:= T#30M;
								END_IF 
								
							ELSE
								Active:=FALSE;
									
								Error:=TRUE;
								ErrorId:=16#0003;
								//{error 'Wrong input values for FB'}
							
								nRunningMode:=0;
								nOperationMode:=0;
								nFbState:=0;
							END_IF
							
							nOperationMode:=2;
						
						ELSIF eLubMode=1 THEN
							
							IF fOutletDosing > 0 AND fLubAmount >= 0 AND fFeedlineGap > 0 THEN
								fTriggerDistance:=fOutletDosing/(fLubAmount*fFeedlineGap);
								fMaxDistanceDrivenTemp:=0;

							ELSE
								Active:=FALSE;
									
								Error:=TRUE;
								ErrorId:=16#0003;
							
								nRunningMode:=0;
								nOperationMode:=0;
								nFbState:=0;
							END_IF
						
							nOperationMode:=3;
						
						ELSIF eLubMode=2 THEN
							
							nOperationMode:=4;
						ELSE
							Active:=FALSE;
									
							Error:=TRUE;
							ErrorId:=16#0003;
						
							nRunningMode:=0;
							nOperationMode:=0;
							nFbState:=0;
						END_IF
						
					
					2: //Lubrication running in time based mode
						CASE nRunningMode OF
							0: //Idle
							
							
							1: //Check if Pump is full
								nRunningMode:=2;
								
							2: //Pumping (1 cycle = 1 OutletDosing per Feedline)
								Busy:=TRUE;
								ObLubOn:=TRUE;
								
								fbTON(IN:=TRUE,PT:=T#7M);	
							
								IF 	fbTON.ET >= T#7M  AND IbLubDone THEN
									fbTON(IN:=FALSE);
									
									ObLubOn:=FALSE;
									Busy:=FALSE;
	
									nRunningMode:=3;
									
								ELSIF fbTon.Q AND NOT IbLubDone THEN
									fbTON(IN:=FALSE);
									ObLubOn:=FALSE;
									
									Busy:=FALSE;
									Active:=FALSE;
									Error:=TRUE;
									ErrorId:=16#0001;
									
									nRunningMode:=0;
									nOperationMode:=0;
									nFbState:=0;		
								END_IF
						
							3: //Waiting (calculated waiting time)
								fbTON(IN:=TRUE,PT:=tPauseTime);
								
								IF fbTON.Q THEN
									fbTON(IN:=FALSE);
									
									nRunningMode:=1;
								END_IF
								
						END_CASE
	
					3: //Lubrication running in distance based mode
						
						CASE nRunningMode OF
							0: //Idle
							
							
							1: //Check if Pump is full	
								nRunningMode:=2;			
								
							2: //Pumping (1 cycle = 1 OutletDosing per Feedline)
								Busy:=TRUE;
								ObLubOn:=TRUE;
								
								fbTON(IN:=TRUE,PT:=T#7M);	
							
								IF 	fbTON.ET > T#7M  AND IbLubDone  THEN
									fbTON(IN:=FALSE);
									
									ObLubOn:=FALSE;
									Busy:=FALSE;
	
									nRunningMode:=3;
									
								ELSIF fbTon.Q AND NOT IbLubDone THEN
									fbTON(IN:=FALSE);
									ObLubOn:=FALSE;
									
									Busy:=FALSE;
									Active:=FALSE;
									Error:=TRUE;
									ErrorId:=16#0001;
									
									nRunningMode:=0;
									nOperationMode:=0;
									nFbState:=0;		
								END_IF
								
								
							3: //Check how far movers have moved
								fbTON(IN:=TRUE,PT:=tPauseTime);
							
								FOR nNumMover:= 1 TO XTSUnitRef.stXtsUnit.stMotion.nAxisCount DO
								
									IF XTSUnitRef.stXtsUnit.stTcIoXtsDrv.stMover[nNumMover].stParameter.fDistanceDriven > fMaxDistanceDriven THEN
										fMaxDistanceDriven:= XTSUnitRef.stXtsUnit.stTcIoXtsDrv.stMover[nNumMover].stParameter.fDistanceDriven;
										nMoverIndex:=nNumMover;
									END_IF
									
								END_FOR	
								
								fMaxDistanceDriven:=fMaxDistanceDriven-fMaxDistanceDrivenTemp;
								
								IF fMaxDistanceDriven >= fTriggerdistance AND fbTon.Q THEN
									fMaxDistanceDrivenTemp:=XTSUnitRef.stXtsUnit.stTcIoXtsDrv.stMover[nMoverIndex].stParameter.fDistanceDriven;
									
									fbTon(In:=FALSE);
									nRunningMode:=1;
								END_IF
										
						END_CASE
			
					4: //Lubrication running in continous mode
					
						CASE nRunningMode OF
							0: //Idle
							
							1: //Pumping (continous)	
								Busy:=TRUE;
								ObLubOn:=TRUE;
								
								fbTON(IN:=TRUE,PT:=T#7M);							
								
								IF 	fbTON.ET >= T#7M  AND IbLubDone THEN
									fbTON(IN:=FALSE);
									
									ObLubOn:=FALSE;
									Busy:=FALSE;
		
									nRunningMode:=2;
									
								ELSIF fbTon.Q AND NOT IbLubDone THEN
									fbTON(IN:=FALSE);
									ObLubOn:=FALSE;
									
									Busy:=FALSE;
									Active:=FALSE;
									Error:=TRUE;
									ErrorId:=16#0001;
									
									nRunningMode:=0;
									nOperationMode:=0;
									nFbState:=0;		
								END_IF
							
							2: //Waiting (calculated waiting time)
								fbTON(IN:=TRUE,PT:=tPauseTime);
								
								IF fbTON.Q THEN
									fbTON(IN:=FALSE);
									
									nRunningMode:=1;
								END_IF
						
						END_CASE
				
				END_CASE
				
		END_CASE	
				
END_CASE

END_FUNCTION_BLOCK

// ---- COMPENENTs/Station/FB_XTS_Station.TcPOU
{attribute 'no_explicit_call' := 'Do not call the body - Stick to OOP'}
FUNCTION_BLOCK FB_XTS_Station EXTENDS FB_CH_Object IMPLEMENTS I_XTS_Station, I_XTS_Station_PLC
VAR
	{attribute 'hide'}
	bInitDone : BOOL;
	{attribute 'hide'}
	bErrorDuringFbInit : BOOL; // Not possible to reset
	{attribute 'hide'}
	ipXtsSystem 				: I_XTS_System_Registration;
	{attribute 'hide'}	
	ipStationInFront 			: I_XTS_Station;
	{attribute 'hide'}	
	ipStationBehinde 			: I_XTS_Station;
	{attribute 'hide'}
	bSuppressDynamicsChange		: BOOL; // Suppress to change the dynamic(Gap+velocity) of passing movers. This is usefull in startup
	{attribute 'hide'}
	fMoverGapAtExit 			: LREAL; // Every mover that leaves or passes the station gets this new gap as a target.
	{attribute 'hide'}
	fMoverVelocityAtExit		: LREAL; // Every mover that leaves or passes the station gets this new velo as a target.	 
	{attribute 'hide'}
	fPositionOnTrack 			: LREAL;
	{attribute 'hide'}
	nMoverQueueSize 			: UINT;
	{attribute 'hide'}
	bReadyToRecvMovers 			: BOOL := TRUE;;
	{attribute 'hide'}
	fTargetPosWindow			: LREAL := 0.05; //[mm]
	{attribute 'hide'}
	tTargetPosMonitoringTime	: TIME := T#0MS;
	{attribute 'hide'}	
	fTrackLentgh 				: LREAL; //[mm]  Modulo
	{attribute 'hide'}
	fbAssignedMovers 			: CHALET_BaseComponents.FB_CH_List;		// List of movers approaching the station
	{attribute 'hide'}
	fbFeedback 					: CHALET_BaseComponents.FB_CH_Feedback(ipSourceInfo := fbSourceInfo);
	{attribute 'hide'}	
	bMoversInPlace : BOOL;
	
	{attribute 'TcInitSymbol'}
	OIDStationInfo : OTCID; //OID of XtsStationInfo object to visualize in Viewer. 0 if not used.
	{attribute 'hide'}
	ipStationInfo : I_TcIoXtsInfoServerInfoStation;
	{attribute 'hide'}
	bUtilityStationInitDone : BOOL;
	
	//Simulation
	{attribute 'hide'}
	fSimulationProcessDuration 	: LREAL; //[s]
	{attribute 'hide'}
	sSimulationTargedStation	: STRING; //LUID of the targed station to automatic send after the duration
	
	
	// ipXtsSystem Is Not Valid at this point, call the konstruktor again in the FB_Init
	{attribute 'hide'}
	fbTrigger 					: FB_XTS_Trigger(ipXtsSystem);
	{attribute 'hide'}
	fbSortedListMoversInQueue	: FB_XTS_Zone(ipXtsSystem);
	
	//Statistic
	{attribute 'hide'}
	fMoverPerMin				: LREAL;
	
END_VAR

METHOD AddMoverToQueue : HRESULT
VAR_INPUT
	ipMover : I_XTS_Mover;
END_VAR
VAR
	ipObject : I_CH_Object;
END_VAR
//Get I_CH_Objekt of mover to put it in to a list.
IF ipMover <> 0 AND_THEN __QUERYINTERFACE(ipMover,ipObject) THEN
	//Add in List of Movers in this station
	THIS^.fbAssignedMovers.AddObject(ipObject);
	
	//Handover information in Mover
	ipMover.ParentStation := (THIS^);

	AddMoverToQueue := S_OK;
ELSE
	AddMoverToQueue := E_FAIL;;	
END_IF
END_METHOD

METHOD ChangePos : HRESULT
VAR_INPUT
	fNewPosOnTrack : LREAL;
END_VAR
VAR
	ipEachMoverInStation : I_XTS_Mover;
	fGapToFirstMoverInQueue, fTargedPos : LREAL;
	nIdx : UDINT;
END_VAR
THIS^.fbFeedback.ActiveCommand := 'ChangePos';
THIS^.fbFeedback.Busy := TRUE;

// Only small changes during system is enabled
IF THIS^.ipXtsSystem.Enabled THEN	
	
	IF fNewPosOnTrack = THIS^.PositionOnTrack THEN
		// failed - same pos
		ChangePos := S_FALSE;
		THIS^.fbFeedback.HR := ChangePos;
		RETURN;
	END_IF	


	// new Position not allowed
	IF fNewPosOnTrack > THIS^.fTrackLentgh THEN
		// failed
		ChangePos := E_FAIL;
		THIS^.fbFeedback.HR := ChangePos;
		RETURN;
	END_IF	
	IF fNewPosOnTrack < 0 THEN
		// failed
		ChangePos := E_FAIL;
		THIS^.fbFeedback.HR := ChangePos;
		RETURN;
	END_IF	
	
	
	IF THIS^.StationBehinde <> 0 AND_THEN fNewPosOnTrack <= THIS^.StationBehinde.PositionOnTrack THEN
		// failed
		ChangePos := E_FAIL;
		THIS^.fbFeedback.HR := ChangePos;
		RETURN;
	END_IF
	IF THIS^.StationsAhead <> 0 AND_THEN fNewPosOnTrack >= THIS^.StationsAhead.PositionOnTrack THEN
		// failed
		ChangePos := E_FAIL;
		THIS^.fbFeedback.HR := ChangePos;
		RETURN;
	END_IF

	
	

	THIS^.fPositionOnTrack := fNewPosOnTrack;
	
	fbTrigger.PositionOnTrack := THIS^.fPositionOnTrack;
	
	// Move the zone 10mm forward to make sure, that an Mover who is enabled at x.01mm is still in range
	fbSortedListMoversInQueue.EndPositionOnTrack := LMOD(lr_Value:=(THIS^.PositionOnTrack + 10.0), lr_Arg:= THIS^.fTrackLentgh); 
	//The zone window is the full system, with one small exception, a window of 0.001mm after the end.  Start and end must not be identical
	fbSortedListMoversInQueue.StartPositionOnTrack := LMOD(lr_Value:=(fbSortedListMoversInQueue.EndPositionOnTrack  + 0.0001), lr_Arg:= THIS^.fTrackLentgh); 
	
	//Redo drawing of station is visu
	THIS^.bUtilityStationInitDone := FALSE;
	
	//Send all movers in this station to new position
	FOR nIdx := 0 TO (XtsParameterlist.MAX_MOVER_PER_SYSTEM-1) DO
		IF ToMover(THIS^.MoversInQueue[nIdx], ipEachMoverInStation) THEN 	
			fTargedPos := fNewPosOnTrack - fGapToFirstMoverInQueue;
			IF fTargedPos < 0 THEN
				fTargedPos := fTargedPos + THIS^.fTrackLentgh;
			END_IF
			ipEachMoverInStation.MoveAbsCA(	fPosition := fTargedPos,
											fVelocity := ipEachMoverInStation.LastCmdTargedVelocity,
											fGap	  := ipEachMoverInStation.LastCmdTargedGap,
											eDirection:= Tc3_Mc3Definitions.MC_DIRECTION.mcDirectionShortestWay	);
											
			fGapToFirstMoverInQueue := fGapToFirstMoverInQueue + ipEachMoverInStation.LastCmdTargedGap;

		ELSE
			EXIT;			
		END_IF
	END_FOR
	
	
	ChangePos := S_OK;


	
// If disabled its allowed to move to any position
ELSIF THIS^.ipXtsSystem.Disabled THEN
	THIS^.fPositionOnTrack := fNewPosOnTrack;
	ChangePos := S_OK;
	
	
	
// During disabling or enabling its not allowed to move the position	
ELSE 
	ChangePos := E_FAIL;;	
END_IF

THIS^.fbFeedback.HR := ChangePos;
END_METHOD

METHOD PROTECTED CheckForStationsSameName : HRESULT
VAR
	fbStationsToCheck : CHALET_BaseComponents.FB_CH_List;
	ipStationToCheck : I_XTS_Station;
END_VAR
VAR_INST
	{attribute 'hide'}	
	fbAlarm : FB_TcAlarm;
END_VAR
//Check for stations on the same position
fbStationsToCheck.Duplicate(THIS^.ipXtsSystem.Stations);

//Clear alarm
fbAlarm.Clear(0,0);

//Remove this station from list
fbStationsToCheck.RemoveObject(THIS^);

// go through the list and search the station in front
fbStationsToCheck.ResetIterator();
WHILE fbStationsToCheck.HasNextObject() DO
	IF ToStation(fbStationsToCheck.GetNextObject(), ipStationToCheck) THEN
		IF ipStationToCheck.PositionOnTrack = THIS^.PositionOnTrack THEN
			fbAlarm.CreateEx(stEventEntry:=TC_EVENTS.CHALET_XTS_Events.DublicateStationNames, ipSourceInfo := THIS^.fbSourceInfo, bWithConfirmation := FALSE);
			fbAlarm.ipArguments.AddStringByValue(THIS^.LUID);
			fbAlarm.Raise(0);
			CheckForStationsSameName := E_FAIL;
			RETURN;
		END_IF	
	END_IF
END_WHILE
END_METHOD

METHOD PROTECTED CheckForStationsSamePos : HRESULT
VAR
	fbStationsToCheck : CHALET_BaseComponents.FB_CH_List;
	ipStationToCheck : I_XTS_Station;
END_VAR
VAR_INST
	{attribute 'hide'}	
	fbAlarm : FB_TcAlarm;
END_VAR
//Check for stations on the same position
fbStationsToCheck.Duplicate(THIS^.ipXtsSystem.Stations);

//Clear alarm
fbAlarm.Clear(0,0);

//Remove this station from list
fbStationsToCheck.RemoveObject(THIS^);

// go through the list and search the station in front
fbStationsToCheck.ResetIterator();
WHILE fbStationsToCheck.HasNextObject() DO
	IF ToStation(fbStationsToCheck.GetNextObject(), ipStationToCheck) THEN
		IF ipStationToCheck.PositionOnTrack = THIS^.PositionOnTrack THEN
			fbAlarm.CreateEx(stEventEntry:=TC_EVENTS.CHALET_XTS_Events.DublicateStationPositions, ipSourceInfo := THIS^.fbSourceInfo, bWithConfirmation := FALSE);
			fbAlarm.ipArguments.AddStringByValue(THIS^.LUID).AddStringByValue(ipStationToCheck.LUID);
			fbAlarm.Raise(0);
			CheckForStationsSamePos := E_FAIL;
			RETURN;
		END_IF	
	END_IF
END_WHILE
END_METHOD

//Call this Methode whith seq 0->99, and wait each step until S_OK is returned
METHOD Configure : HRESULT
VAR_INPUT
	nSeq : UINT; //0->100
END_VAR
VAR

END_VAR
VAR_INST
	{attribute 'hide'}	
	fbInvalideStationPositionAlarm : FB_TcAlarm;
END_VAR
CASE nSeq OF

	1: // Reset Config-Errors
		fbInvalideStationPositionAlarm.Clear(0,0);
		

	2: //Check for valide Data
		IF 	THIS^.ipXtsSystem = 0 OR 
			THIS^.ipXtsSystem.Environment = 0 OR
			THIS^.ipXtsSystem.Stations = 0 THEN
				Configure := E_FAIL;
		END_IF	
			
	
	3: //Store some data
		THIS^.fTrackLentgh := THIS^.ipXtsSystem.TrackLength;
		IF THIS^.fTrackLentgh <= 0 THEN
			Configure := E_FAIL;
		END_IF
		
		
	10: //Station position on track is larger than CA-Group track length
		IF THIS^.PositionOnTrack > THIS^.fTrackLentgh THEN
			fbInvalideStationPositionAlarm.CreateEx(stEventEntry:=TC_EVENTS.CHALET_XTS_Events.StationPositionLargerAsTrack, ipSourceInfo := THIS^.fbSourceInfo, bWithConfirmation := FALSE);
			fbInvalideStationPositionAlarm.Raise(0);
			Configure := E_FAIL;
		END_IF

		
	20: //Error if two stations have the same LUID
		Configure := THIS^.CheckForStationsSameName();
		
				
	30: //Error if two stations have the same position on track
		Configure := THIS^.CheckForStationsSamePos();
		
		
	40: //Get Station in Front
		Configure := THIS^.GetStationAhead();
	
			
				
	50: //Get Station in Back
		Configure := THIS^.GetStationBehinde();
			
		
	60: // Config trigger fb
		THIS^.fbTrigger.ListOfMoversToCheck := THIS^.ipXtsSystem.Movers;
		THIS^.fbTrigger.PositionOnTrack := THIS^.PositionOnTrack;
		THIS^.fbTrigger.TriggerDirection := MC_Positive_Direction;
		Configure := THIS^.fbTrigger.Initialize();		
		
	70: // Config window fb		
		// Use the zone to sort all movers in this queue depending on the distance to targed in an output array.
		// Move the zone 10mm forward to make sure, that an Mover who is enabled at x.01mm is still in range
		fbSortedListMoversInQueue.EndPositionOnTrack := LMOD(lr_Value:=(THIS^.PositionOnTrack + 10.0), lr_Arg:= THIS^.fTrackLentgh); 
		//The zone window is the full system, with one small exception, a window of 0.001mm after the end.  Start and end must not be identical
		fbSortedListMoversInQueue.StartPositionOnTrack := LMOD(lr_Value:=(fbSortedListMoversInQueue.EndPositionOnTrack  + 0.0001), lr_Arg:= THIS^.fTrackLentgh); 
		fbSortedListMoversInQueue.ListOfMoversToCheck := THIS^.fbAssignedMovers;
		Configure := THIS^.fbSortedListMoversInQueue.Initialize();	
		

		
	80: //Redo drawing of station is visu
		THIS^.bUtilityStationInitDone := FALSE;	

	100..CHALET_BaseComponents.GVL_Datatypes.cMaxUint: 
		// 100..MaxUint -> Invalide input
		Configure := E_FAIL;
		
	ELSE 
		//If an step is not defind/used return ok
		Configure := S_OK;
END_CASE
END_METHOD

{attribute 'monitoring':='call'}
PROPERTY CtsEmptySpaceInQueue : UDINT
GET
//Handle UINT Overflow
IF THIS^.fbAssignedMovers.Size >= THIS^.nMoverQueueSize THEN
	CtsEmptySpaceInQueue := 0;
ELSE 
	CtsEmptySpaceInQueue := THIS^.nMoverQueueSize - THIS^.fbAssignedMovers.Size;
END_IF
END_GET
END_PROPERTY

{attribute 'monitoring':='call'}
PROPERTY CtsMoversInQueue : UDINT
GET
CtsMoversInQueue := THIS^.fbAssignedMovers.Size;
END_GET
END_PROPERTY

METHOD DeleteMoversQueue : HRESULT
VAR
	ipTempMover : I_XTS_Mover;
END_VAR
//Delete intormation in linked mover
fbAssignedMovers.ResetIterator();
WHILE fbAssignedMovers.HasNextObject() DO
	IF ToMover(fbAssignedMovers.GetNextObject(),ipTempMover) THEN
		ipTempMover.ParentStation := 0;
	END_IF	
END_WHILE

//Clear list
THIS^.fbAssignedMovers.Clear();
DeleteMoversQueue := S_OK;
END_METHOD

METHOD FB_init : BOOL
VAR_INPUT
	bInitRetains : BOOL; // if TRUE, the retain variables are initialized (warm start / cold start)
	bInCopyCode : BOOL;  // if TRUE, the instance afterwards gets moved into the copy code (online change)
	
	ipXtsSystem 			: I_XTS_System_Registration; //Interface to XTS system object
	fPositionOnTrack 		: LREAL;	//[mm]
	sUniqueName				: STRING;	//expl.:'Loading'
	nMoverQueueSize 		: UINT;		//[cts]
	
	//Dynamik at exit of station
	fMoverGapAtExit 		: LREAL;	//[mm]
	fMoverVelocityAtExit 	: LREAL;	//[mm/s]

END_VAR
VAR_INST
	{attribute 'hide'}
	bFBInitCalledOnce : BOOL; //Do the following code once during start up and not during onlinechange
END_VAR
//Do the following code once during start up and not during onlinechange
IF NOT bFBInitCalledOnce THEN 
	
	//Regristrate object in System
	IF ipXtsSystem <> 0 THEN
		ipXtsSystem.RegisterStation(THIS^);
		THIS^.ipXtsSystem := ipXtsSystem;
	END_IF

	//"" is maybe entered in an waiting or dynamic station and the name is not important
	IF sUniqueName <> '' THEN 
		THIS^.fbSourceInfo.sName := sUniqueName;
	ELSE
		sUniqueName := THIS^.fbSourceInfo.sName;
	END_IF
	
	THIS^.fMoverGapAtExit := fMoverGapAtExit;
	THIS^.fMoverVelocityAtExit := fMoverVelocityAtExit;
	THIS^.nMoverQueueSize := nMoverQueueSize;
	THIS^.fPositionOnTrack := fPositionOnTrack;
	
	THIS^.fbTrigger.FB_init(FALSE,FALSE, ipXtsSystem);
	THIS^.fbSortedListMoversInQueue.FB_init(FALSE,FALSE, ipXtsSystem);

END_IF

bFBInitCalledOnce := TRUE;
END_METHOD

(*The _ PLC interface provides the user with a simplified interface for commanding between the stations. Sometimes, however, this is not enough. 
Either you get the corresponding interface with the __Queryinterface or you can get full access with this property.*)
PROPERTY FullAccess : I_XTS_Station
GET
FullAccess := (THIS^);
END_GET
END_PROPERTY

METHOD PROTECTED GetStationAhead : HRESULT
VAR
	fbStationsToCheck	: CHALET_BaseComponents.FB_CH_List;
	ipStationToCheck 	: I_XTS_Station;	
	bTrackIsRing			: BOOL;

	fTempDistBetween 	: LREAL;
	
	fFoundDistBetween 	: LREAL := CHALET_BaseComponents.GVL_Datatypes.cMaxLreal;
	ipFoundStation		: I_XTS_Station;
END_VAR
//Clear
THIS^.ipStationInFront := 0;

//get new lisat of stations
fbStationsToCheck.Duplicate(THIS^.ipXtsSystem.Stations);

bTrackIsRing := THIS^.ipXtsSystem.Environment.TrackIsRing;


//Remove this station from list
fbStationsToCheck.RemoveObject(THIS^);

// go through the list and search the station in front
fbStationsToCheck.ResetIterator();
WHILE fbStationsToCheck.HasNextObject() DO
	IF ToStation(fbStationsToCheck.GetNextObject(), ipStationToCheck) THEN
		
		IF NOT bTrackIsRing AND (ipStationToCheck.PositionOnTrack < THIS^.PositionOnTrack) THEN
			// Skip this station if behinde and not a closed loop
			CONTINUE;
		END_IF
		
		// calc distance to position in positive direction
		fTempDistBetween := F_GetDistToPosModulo(	fActualPosition := THIS^.PositionOnTrack,
													fTargedPosition := ipStationToCheck.PositionOnTrack, 
													fModulo := THIS^.fTrackLentgh);

		// check if Station is closer then last one - store
		IF fFoundDistBetween > fTempDistBetween THEN 
			fFoundDistBetween := fTempDistBetween;
			THIS^.ipStationInFront := ipStationToCheck;
		END_IF
		
	END_IF
END_WHILE
END_METHOD

METHOD PROTECTED GetStationBehinde : HRESULT
VAR
	fbStationsToCheck	: CHALET_BaseComponents.FB_CH_List;
	ipStationToCheck 	: I_XTS_Station;	

END_VAR
//Clear
THIS^.ipStationBehinde := 0;

//get new lisat of stations
fbStationsToCheck.Duplicate(THIS^.ipXtsSystem.Stations);

//Remove this station from list
fbStationsToCheck.RemoveObject(THIS^);

// go through the list and search the station in front
fbStationsToCheck.ResetIterator();
WHILE fbStationsToCheck.HasNextObject() DO
	IF ToStation(fbStationsToCheck.GetNextObject(), ipStationToCheck) THEN
		
		IF ipStationToCheck.StationsAhead.LUID = THIS^.LUID THEN
			//FOUND
			THIS^.ipStationBehinde := ipStationToCheck;
			RETURN;
		END_IF
		
	END_IF
END_WHILE
END_METHOD

{attribute 'monitoring':='call'}
PROPERTY HR : HRESULT
GET
HR := fbFeedback.hr;
END_GET
END_PROPERTY

METHOD Initialize : HRESULT
VAR
	nLoopIndex : UDINT;
	nNbOfStationsChecked : UDINT;
	//ipThisStation, ipTempStation, ipStationInFrontTemp : I_XTS_Station;
	bErrorStationInFrontNotFound, bErrorStationBehindeNotFound : BOOL;
END_VAR
VAR_INST
	//This error cannot be reset. Requires a reset cold
	{attribute 'hide'}	
	fbInitError : FB_TcAlarm;
	{attribute 'hide'}	
	fbMissingInterfaceAlarm : FB_TcAlarm;

END_VAR
fbFeedback.ActiveCommand := 'Initialize';
fbFeedback.hr := S_PENDING;	

